// TIA Portal V15.1 export
// export: Created 2024-09-12T07:42:50.9677284Z, ExportSetting WithDefaults, DisplayName Totally Integrated Automation Portal, DisplayVersion V15.1 Update 5, DisplayName TIA Portal Openness, DisplayVersion V15.1 Update 5, DisplayName SINAMICS Startdrive Advanced, DisplayVersion V15.1, DisplayName G130, G150, S120, S150, SINAMICS MV, S210, DisplayVersion V15.1, DisplayName G110M, G120, G120C, G120D, G120P, DisplayVersion V15.1, DisplayName STEP 7 Professional, DisplayVersion V15.1 Update 5, DisplayName STEP 7 Safety, DisplayVersion V15.1, DisplayName WinCC Professional, DisplayVersion V15.1 Update 5, DisplayName SIMATIC Visualization Architect, DisplayVersion V15.1
FUNCTION_BLOCK "LSystemVarS7-1500"   // FB2204, FBD
TITLE = LSystemVarS7-1500
{ S7_Optimized_Access := 'TRUE' }
AUTHOR : VCC
FAMILY : Control
VERSION : 0.1
// =============================================================================
// This module is used to handle system variables such as Blink, Pulse, 
// ,Cycletime and CPU System Time used in timer modules.
// =============================================================================
// stored: AutoNumber false, IsIECCheckEnabled false, IsRetainMemResEnabled false, MemoryReserve 100, SetENOAutomatically False, UDAEnableTagReadback false
   VAR_INPUT
      I_OB1Cycletime { ExternalAccessible := 'False'; ExternalVisible := 'False'; ExternalWritable := 'False'} : Int;   // Cycle time of previous OB1 scan (milliseconds)
      I_PLCLADDR { ExternalAccessible := 'False'; ExternalVisible := 'False'; ExternalWritable := 'False'} : HW_IO;   // Hardware I/O
      I_DateTime { ExternalAccessible := 'False'; ExternalVisible := 'False'; ExternalWritable := 'False'} : Date_And_Time;   // Date and time
      I_AlarmResetPB { ExternalAccessible := 'False'; ExternalVisible := 'False'; ExternalWritable := 'False'} : Bool;   // Alarm reset pushbutton is activated / Alarm Reset Pushbutton is Activated
      I_EnableAlarm { ExternalAccessible := 'False'; ExternalVisible := 'False'; ExternalWritable := 'False'} : Bool := TRUE;   // Enable alarm from upper level / Enable Alarm from upper level
      C_HMIBtnResetSeqResetTM { ExternalAccessible := 'False'; ExternalVisible := 'False'; ExternalWritable := 'False'} : Bool;   // HMI buttons ResetSeq & ResetTM (0=Buttons are separate ; 1=Buttons are common)
      C_PlantId { ExternalAccessible := 'False'; ExternalVisible := 'False'; ExternalWritable := 'False'} : Int;   // Plant Identification (1=VCT, 2=VCBC, 3=VCG, 4=VCCH, 5=VCCD, 6=VCDQ, 7=AELQ, 8=PSCD)
      C_ShopId { ExternalAccessible := 'False'; ExternalVisible := 'False'; ExternalWritable := 'False'} : Int;   // Shop Identification (10=A-shop, 11=B-shop, 12=C-shop, 13=D-shop, 19=Stamping)
      C_LanguageChangeTimeToDefault { ExternalAccessible := 'False'; ExternalVisible := 'False'; ExternalWritable := 'False'} : Time := T#60m;   // Time to change back to default language. Connect T#0M to disable timer
   END_VAR
   VAR_OUTPUT
      O_AlarmABCondition { ExternalAccessible := 'False'; ExternalVisible := 'False'; ExternalWritable := 'False'} : Bool;   // Alarm AB condition / Alarm AB Condition
      O_AlarmA { ExternalAccessible := 'False'; ExternalVisible := 'False'; ExternalWritable := 'False'} : Bool;   // Summation Alarm A. / Alarm A
      O_AlarmB { ExternalAccessible := 'False'; ExternalVisible := 'False'; ExternalWritable := 'False'} : Bool;   // Summation Alarm B. / Alarm B
      O_AlarmC { ExternalAccessible := 'False'; ExternalVisible := 'False'; ExternalWritable := 'False'} : Bool;   // Summation Alarm C. / Alarm C.
      O_AlarmD { ExternalAccessible := 'False'; ExternalVisible := 'False'; ExternalWritable := 'False'} : Bool;   // Summation Alarm D. / Alarm D.
      O_AlarmWord { ExternalAccessible := 'False'; ExternalVisible := 'False'; ExternalWritable := 'False'} : DWord;   // Alarm Word
      O_SystemTime { ExternalAccessible := 'False'; ExternalVisible := 'False'; ExternalWritable := 'False'} : Array[0..2] of DWord;   // System Time
   END_VAR
   VAR_IN_OUT
      IO_Alarm : "Alarm";   // Alarm
      IO_SetDateTime { ExternalAccessible := 'False'; ExternalVisible := 'False'; ExternalWritable := 'False'} : Bool;   // Set date and time
      H_HMI : "H_HMI";   // HMI
      "H_SystemVarS7-1500" : "H_SystemVarS7-1500";   // Animation
      C_SwedishLanguage { ExternalAccessible := 'False'; ExternalVisible := 'False'; ExternalWritable := 'False'} : Bool;   // Swedisch Language
      C_DutchLanguage { ExternalAccessible := 'False'; ExternalVisible := 'False'; ExternalWritable := 'False'} : Bool;   // Dutch Language
      C_EnglishLanguage { ExternalAccessible := 'False'; ExternalVisible := 'False'; ExternalWritable := 'False'} : Bool;   // English Language
      C_ChineseLanguage { ExternalAccessible := 'False'; ExternalVisible := 'False'; ExternalWritable := 'False'} : Bool;   // Chinese Language
      C_ScreenSaverEnable { ExternalAccessible := 'False'; ExternalVisible := 'False'; ExternalWritable := 'False'} : Bool;   // Screen Saver HMI Panels
   END_VAR
   VAR
      AB_FALSE { ExternalAccessible := 'False'; ExternalVisible := 'False'; ExternalWritable := 'False'} : Bool;   // Systemvariabel Logiskt Resultat "TRUE" = "FALSE" / System Variable Logic Result TRUE Should Be FALSE
      AB_TRUE { ExternalAccessible := 'False'; ExternalVisible := 'False'; ExternalWritable := 'False'} : Bool;   // Systemvariabel Logiskt Resultat "FALSE" = "TRUE" / System Variable Logic Result FALSE Should Be TRUE
      AD_OB40 { ExternalAccessible := 'False'; ExternalVisible := 'False'; ExternalWritable := 'False'} : Bool;   // 0000: Hardware Interrupt 0 / Hardware Interrupt / Hårdvaru Interrupt
      AD_OB80 { ExternalAccessible := 'False'; ExternalVisible := 'False'; ExternalWritable := 'False'} : Bool;   // 0000: Cycle Time Fault / Cycle Time Error / Cykeltidsfel
      AD_OB81 { ExternalAccessible := 'False'; ExternalVisible := 'False'; ExternalWritable := 'False'} : Bool;   // 0000: Power Supply Fault / Error On Power Supply / Fel På Spänningsaggregat
      AD_OB82 { ExternalAccessible := 'False'; ExternalVisible := 'False'; ExternalWritable := 'False'} : Bool;   // 0000: I/O Point Fault 1 / I/O Error / I/O Fel
      AD_OB83 { ExternalAccessible := 'False'; ExternalVisible := 'False'; ExternalWritable := 'False'} : Bool;   // 0000: I/O Point Fault 2 / I/O Error / I/O Fel
      AD_OB84 { ExternalAccessible := 'False'; ExternalVisible := 'False'; ExternalWritable := 'False'} : Bool;   // 0000: CPU Fault / CPU Error / CPU Fel
      AD_OB85 { ExternalAccessible := 'False'; ExternalVisible := 'False'; ExternalWritable := 'False'} : Bool;   // 0000: OB Not Loaded Fault / I/O Access Error / I/O Access Fel
      AD_OB86 { ExternalAccessible := 'False'; ExternalVisible := 'False'; ExternalWritable := 'False'} : Bool;   // 0000: Loss of Rack Fault / CPU Rack Error / CPU Rack Fel
      AD_OB87 { ExternalAccessible := 'False'; ExternalVisible := 'False'; ExternalWritable := 'False'} : Bool;   // 0000: Communication Fault / Communication Error / Kommunikationsfel
      AD_OB100 { ExternalAccessible := 'False'; ExternalVisible := 'False'; ExternalWritable := 'False'} : Bool;   // 0000: Complete Restart / CPU Warm Restart / CPU Varm Omstart
      AD_OB101 { ExternalAccessible := 'False'; ExternalVisible := 'False'; ExternalWritable := 'False'} : Bool;   // Hot Restart / Omstart
      AD_OB102 { ExternalAccessible := 'False'; ExternalVisible := 'False'; ExternalWritable := 'False'} : Bool;   // 0000: Cold Restart / Cold Restart / Omstart
      AB_OB121 { ExternalAccessible := 'False'; ExternalVisible := 'False'; ExternalWritable := 'False'} : Bool;   // 0000: Programming Error / Programming Error / Programmeringsfel
      AD_OB122 { ExternalAccessible := 'False'; ExternalVisible := 'False'; ExternalWritable := 'False'} : Bool;   // 0000: Module Access Error / I/O Module Access Error / I/O Modul Access Fel
      AD_Forced { ExternalAccessible := 'False'; ExternalVisible := 'False'; ExternalWritable := 'False'} : Bool;   // 0000: Forced I/O in CPU / I/O Are Forced In CPU / I/O Är Forcerade I CPU
      AD_Error { ExternalAccessible := 'False'; ExternalVisible := 'False'; ExternalWritable := 'False'} : Bool;   // Error In Software Or Hardware Check Diagnostics / Fel I Mjukvara Eller Hårdvara Kontrollera Diagnostik
      AD_Warning { ExternalAccessible := 'False'; ExternalVisible := 'False'; ExternalWritable := 'False'} : Bool;   // Warning In Software Or Hardware Check Diagnostics / Varning I Mjukvara Eller Hårdvara Kontrollera Diagnostik
      AE_CalibrationMovUnit { ExternalAccessible := 'False'; ExternalVisible := 'False'; ExternalWritable := 'False'} : Bool;   // Kalibrering MovUnit's Utförd / Info -> Redo Overtime calibration MovUnit / Calibration MovUnit's Executed
      AE_CalibrationTransfers { ExternalAccessible := 'False'; ExternalVisible := 'False'; ExternalWritable := 'False'} : Bool;   // Kalibrering MovUnit's Utförd / Info -> Redo Overtime calibration Transfers / Calibration MovUnit's Executed
      AE_Simulation { ExternalAccessible := 'False'; ExternalVisible := 'False'; ExternalWritable := 'False'} : Bool;   // Kalibrering MovUnit's Utförd / Info -> Simulation is active / Calibration MovUnit's Executed
      PulseBlink0_1s { ExternalAccessible := 'False'; ExternalVisible := 'False'; ExternalWritable := 'False'} : Bool;   // Help memory for pulse 0.1s
      PulseBlink0_2s { ExternalAccessible := 'False'; ExternalVisible := 'False'; ExternalWritable := 'False'} : Bool;   // Help memory for pulse 0.2s
      PulseBlink0_4s { ExternalAccessible := 'False'; ExternalVisible := 'False'; ExternalWritable := 'False'} : Bool;   // Help memory for pulse 0.4s
      PulseBlink0_5s { ExternalAccessible := 'False'; ExternalVisible := 'False'; ExternalWritable := 'False'} : Bool;   // Help memory for pulse 0.5s
      PulseBlink0_8s { ExternalAccessible := 'False'; ExternalVisible := 'False'; ExternalWritable := 'False'} : Bool;   // Help memory for pulse 0.8s
      PulseBlink1_0s { ExternalAccessible := 'False'; ExternalVisible := 'False'; ExternalWritable := 'False'} : Bool;   // Help memory for pulse 1.0s
      PulseBlink1_6s { ExternalAccessible := 'False'; ExternalVisible := 'False'; ExternalWritable := 'False'} : Bool;   // Help memory for pulse 1.6s
      PulseBlink2_0s { ExternalAccessible := 'False'; ExternalVisible := 'False'; ExternalWritable := 'False'} : Bool;   // Help memory for pulse 2.0s
      AlarmA { ExternalAccessible := 'False'; ExternalVisible := 'False'; ExternalWritable := 'False'} : Bool;   // Summation Alarm A / Alarm A
      AlarmB { ExternalAccessible := 'False'; ExternalVisible := 'False'; ExternalWritable := 'False'} : Bool;   // Summation Alarm B / Alarm B
      AlarmC { ExternalAccessible := 'False'; ExternalVisible := 'False'; ExternalWritable := 'False'} : Bool;   // Summation Alarm C / Alarm C
      AlarmD { ExternalAccessible := 'False'; ExternalVisible := 'False'; ExternalWritable := 'False'} : Bool;   // Summation Alarm D / Alarm D
      AlarmOB40 { ExternalAccessible := 'False'; ExternalVisible := 'False'; ExternalWritable := 'False'} : Bool;   // Alarm OB40
      AlarmOB80 { ExternalAccessible := 'False'; ExternalVisible := 'False'; ExternalWritable := 'False'} : Bool;   // Alarm OB80
      AlarmOB81 { ExternalAccessible := 'False'; ExternalVisible := 'False'; ExternalWritable := 'False'} : Bool;   // Alarm OB81
      AlarmOB82 { ExternalAccessible := 'False'; ExternalVisible := 'False'; ExternalWritable := 'False'} : Bool;   // Alarm OB82
      AlarmOB83 { ExternalAccessible := 'False'; ExternalVisible := 'False'; ExternalWritable := 'False'} : Bool;   // Alarm OB83
      AlarmOB84 { ExternalAccessible := 'False'; ExternalVisible := 'False'; ExternalWritable := 'False'} : Bool;   // Alarm OB84
      AlarmOB85 { ExternalAccessible := 'False'; ExternalVisible := 'False'; ExternalWritable := 'False'} : Bool;   // Alarm OB85
      AlarmOB86 { ExternalAccessible := 'False'; ExternalVisible := 'False'; ExternalWritable := 'False'} : Bool;   // Alarm OB86
      AlarmOB87 { ExternalAccessible := 'False'; ExternalVisible := 'False'; ExternalWritable := 'False'} : Bool;   // Alarm OB87
      AlarmOB100 { ExternalAccessible := 'False'; ExternalVisible := 'False'; ExternalWritable := 'False'} : Bool;   // Alarm OB100
      AlarmOB101 { ExternalAccessible := 'False'; ExternalVisible := 'False'; ExternalWritable := 'False'} : Bool;   // Alarm OB101
      AlarmOB102 { ExternalAccessible := 'False'; ExternalVisible := 'False'; ExternalWritable := 'False'} : Bool;   // Alarm OB102
      AlarmOB121 { ExternalAccessible := 'False'; ExternalVisible := 'False'; ExternalWritable := 'False'} : Bool;   // Alarm OB121
      AlarmOB122 { ExternalAccessible := 'False'; ExternalVisible := 'False'; ExternalWritable := 'False'} : Bool;   // Alarm OB122
      Edge { ExternalAccessible := 'False'; ExternalVisible := 'False'; ExternalWritable := 'False'} : Array[0..15] of Bool;   // Edge
      MemOB40Execution { ExternalAccessible := 'False'; ExternalVisible := 'False'; ExternalWritable := 'False'} : Int;   // Memorisation previous value number of executuons of OB40
      MemOB80Execution { ExternalAccessible := 'False'; ExternalVisible := 'False'; ExternalWritable := 'False'} : Int;   // Memorisation previous value number of executuons of OB80
      MemOB81Execution { ExternalAccessible := 'False'; ExternalVisible := 'False'; ExternalWritable := 'False'} : Int;   // Memorisation previous value number of executuons of OB81
      MemOB82Execution { ExternalAccessible := 'False'; ExternalVisible := 'False'; ExternalWritable := 'False'} : Int;   // Memorisation previous value number of executuons of OB82
      MemOB83Execution { ExternalAccessible := 'False'; ExternalVisible := 'False'; ExternalWritable := 'False'} : Int;   // Memorisation previous value number of executuons of OB83
      MemOB84Execution { ExternalAccessible := 'False'; ExternalVisible := 'False'; ExternalWritable := 'False'} : Int;   // Memorisation previous value number of executuons of OB84
      MemOB85Execution { ExternalAccessible := 'False'; ExternalVisible := 'False'; ExternalWritable := 'False'} : Int;   // Memorisation previous value number of executuons of OB85
      MemOB86Execution { ExternalAccessible := 'False'; ExternalVisible := 'False'; ExternalWritable := 'False'} : Int;   // Memorisation previous value number of executuons of OB86
      MemOB87Execution { ExternalAccessible := 'False'; ExternalVisible := 'False'; ExternalWritable := 'False'} : Int;   // Memorisation previous value number of executuons of OB87
      MemOB100Execution { ExternalAccessible := 'False'; ExternalVisible := 'False'; ExternalWritable := 'False'} : Int;   // Memorisation previous value number of executuons of OB100
      MemOB101Execution { ExternalAccessible := 'False'; ExternalVisible := 'False'; ExternalWritable := 'False'} : Int;   // Memorisation previous value number of executuons of OB101
      MemOB102Execution { ExternalAccessible := 'False'; ExternalVisible := 'False'; ExternalWritable := 'False'} : Int;   // Memorisation previous value number of executuons of OB102
      MemOB121Execution { ExternalAccessible := 'False'; ExternalVisible := 'False'; ExternalWritable := 'False'} : Int;   // Memorisation previous value number of executuons of OB121
      MemOB122Execution { ExternalAccessible := 'False'; ExternalVisible := 'False'; ExternalWritable := 'False'} : Int;   // Memorisation previous value number of executuons of OB122
      HMICmd_CalibrateMovUnits { ExternalAccessible := 'False'; ExternalVisible := 'False'; ExternalWritable := 'False'} : Bool;   // HMI Command - Calibrate Move Units
      HMICmd_CalibrateTransfers { ExternalAccessible := 'False'; ExternalVisible := 'False'; ExternalWritable := 'False'} : Bool;   // HMI Command - Calibrate Transfers
      HMICmd_Simulation { ExternalAccessible := 'False'; ExternalVisible := 'False'; ExternalWritable := 'False'} : Bool;   // HMI Command - Simulation
      HMICmd_DisableIOAlarm { ExternalAccessible := 'False'; ExternalVisible := 'False'; ExternalWritable := 'False'} : Bool;   // HMI Command - Disable IO Alarm
      ActualScanTimeOB1 { ExternalAccessible := 'False'; ExternalVisible := 'False'; ExternalWritable := 'False'} : LTime;   // Animation / FB
      LongestScanTimeOB1 { ExternalAccessible := 'False'; ExternalVisible := 'False'; ExternalWritable := 'False'} : LTime;   // Animation / FB
      EnableAlarm { ExternalAccessible := 'False'; ExternalVisible := 'False'; ExternalWritable := 'False'} : Bool := TRUE;   // Enable alarm from upper level / Enable Alarm from upper level
      LanguageChangeToDefault { ExternalAccessible := 'False'; ExternalVisible := 'False'; ExternalWritable := 'False'} : Bool;   // Change language back to default
      LanguageDefaultTime { ExternalAccessible := 'False'; ExternalVisible := 'False'; ExternalWritable := 'False'} : DInt;   // Language to default time running value
      DBnr { ExternalAccessible := 'False'; ExternalVisible := 'False'; ExternalWritable := 'False'} : Int;   // HMI DB number
      TimerOffOB40 { ExternalAccessible := 'False'; ExternalVisible := 'False'; ExternalWritable := 'False'} : TOF_TIME;   // FB / Timer
      TimerOffOB80 { ExternalAccessible := 'False'; ExternalVisible := 'False'; ExternalWritable := 'False'} : TOF_TIME;   // FB / Timer
      TimerOffOB81 { ExternalAccessible := 'False'; ExternalVisible := 'False'; ExternalWritable := 'False'} : TOF_TIME;   // FB / Timer
      TimerOffB83 { ExternalAccessible := 'False'; ExternalVisible := 'False'; ExternalWritable := 'False'} : TOF_TIME;   // FB / Timer
      TimerOffOB84 { ExternalAccessible := 'False'; ExternalVisible := 'False'; ExternalWritable := 'False'} : TOF_TIME;   // FB / Timer
      TimerOffOB85 { ExternalAccessible := 'False'; ExternalVisible := 'False'; ExternalWritable := 'False'} : TOF_TIME;   // FB / Timer
      TimerOffOB86 { ExternalAccessible := 'False'; ExternalVisible := 'False'; ExternalWritable := 'False'} : TOF_TIME;   // FB / Timer
      TimerOffOB87 { ExternalAccessible := 'False'; ExternalVisible := 'False'; ExternalWritable := 'False'} : TOF_TIME;   // FB / Timer
      TimerOffOB100 { ExternalAccessible := 'False'; ExternalVisible := 'False'; ExternalWritable := 'False'} : TOF_TIME;   // FB / Timer
      TimerOffOB101 { ExternalAccessible := 'False'; ExternalVisible := 'False'; ExternalWritable := 'False'} : TOF_TIME;   // FB / Timer
      TimerOffOB102 { ExternalAccessible := 'False'; ExternalVisible := 'False'; ExternalWritable := 'False'} : TOF_TIME;   // FB / Timer
      TimerOffOB121 { ExternalAccessible := 'False'; ExternalVisible := 'False'; ExternalWritable := 'False'} : TOF_TIME;   // FB / Timer
      TimerOffOB122 { ExternalAccessible := 'False'; ExternalVisible := 'False'; ExternalWritable := 'False'} : TOF_TIME;   // FB / Timer
      TimerCalibrationMovUnit { ExternalAccessible := 'False'; ExternalVisible := 'False'; ExternalWritable := 'False'} : TOF_TIME;   // Timer
      TimerCalibrationTransfers { ExternalAccessible := 'False'; ExternalVisible := 'False'; ExternalWritable := 'False'} : TOF_TIME;   // Timer
      TimerGlobalSelAutoMode { ExternalAccessible := 'False'; ExternalVisible := 'False'; ExternalWritable := 'False'} : TON_TIME;   // Timer
      TimerGlobalSelManualMode { ExternalAccessible := 'False'; ExternalVisible := 'False'; ExternalWritable := 'False'} : TON_TIME;   // Timer
      _GetIMData { ExternalAccessible := 'False'; ExternalVisible := 'False'; ExternalWritable := 'False'} : Get_IM_Data;   // FB
      _DlyErr { ExternalAccessible := 'False'; ExternalVisible := 'False'; ExternalWritable := 'False'} : TON_TIME;   // Timer
      _DlyWarning { ExternalAccessible := 'False'; ExternalVisible := 'False'; ExternalWritable := 'False'} : TON_TIME;   // Timer
      _ScreenSaverHMI { ExternalAccessible := 'False'; ExternalVisible := 'False'; ExternalWritable := 'False'} : "LTimer";   // Timer
      _LanguageDefault { ExternalAccessible := 'False'; ExternalVisible := 'False'; ExternalWritable := 'False'} : TON_TIME;   // Timer
      _LToggleDisableIOAlarm { ExternalAccessible := 'False'; ExternalVisible := 'False'; ExternalWritable := 'False'} : "LToggle";   // FB
   END_VAR
   VAR_TEMP
      TmpSystemTime : DTL;   // Temporary DTL Day / Temp
      TmpSystemHourMin : UInt;   // Temp
      TmpRetValTime : Int;   // Temp RetVal of TD_SYS_T / Temp
      TmpWeekday : Int;   // Temporary weekday / Temp
      TmpResult : Int;   // Temporary result / Temp
      SetClkRet : Int;   // Return value / Temp
      ReadSysstData : Struct   // data read / Temp
         "STOP/RUN" : Int;   // Stop, Run
         ERROR : Int;   // Error
         MAINT : Int;   // Maintanance
      END_STRUCT;
      LED1C1On : Bool;   // LED 1 color 1: Green on
      LED1C1Blink : Bool;   // LED 1 color 1: Green blinking
      LED1C2On : Bool;   // LED 1 color 2: Yellow on
      LED1C2Blink : Bool;   // LED 1 color 2: Yellow blinking
      LED2C1On : Bool;   // LED 2 color 1: Red on
      LED2C1Blink : Bool;   // LED 2 color 1: Red blinking
      LED3C1On : Bool;   // LED 3 color 1: Yellow on
      LED3C1Blink : Bool;   // LED 3 color 1: Yellow blinking
      IMData : IM0_Data;   // Temp
      tNotUsedDInt : DInt;   // Temp
   END_VAR
   VAR_TEMP   // added for the SCL form of the ladder/FBD networks
      _w1 : Bool;
      _w2 : Bool;
      _w3 : Bool;
      _w4 : Bool;
      _w5 : Bool;
   END_VAR
BEGIN

REGION Network 1: **** 1 - Inputs **** Extract HMI Commands
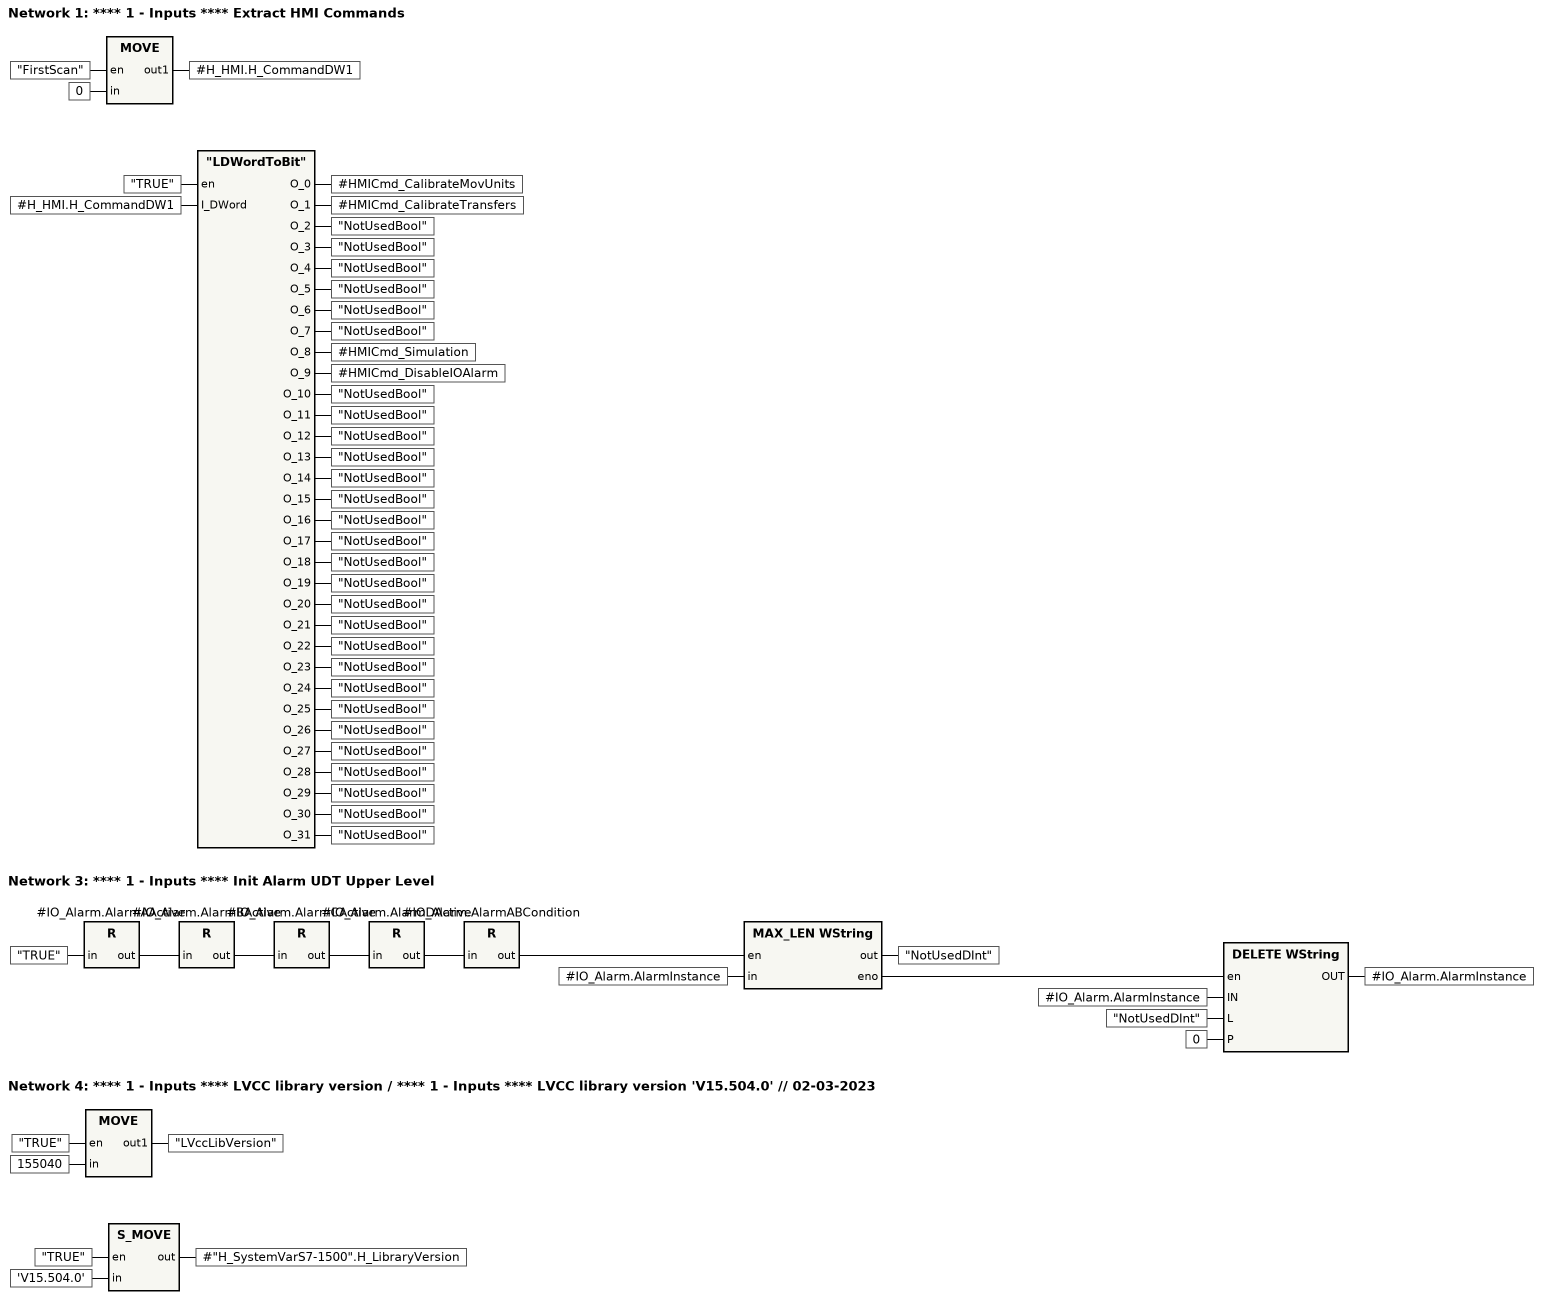
   IF "FirstScan" THEN #H_HMI.H_CommandDW1 := 0; END_IF;
   IF "TRUE" THEN
       "LDWordToBit"(I_DWord := #H_HMI.H_CommandDW1,
                     O_0 => #HMICmd_CalibrateMovUnits,
                     O_1 => #HMICmd_CalibrateTransfers,
                     O_2 => "NotUsedBool",
                     O_3 => "NotUsedBool",
                     O_4 => "NotUsedBool",
                     O_5 => "NotUsedBool",
                     O_6 => "NotUsedBool",
                     O_7 => "NotUsedBool",
                     O_8 => #HMICmd_Simulation,
                     O_9 => #HMICmd_DisableIOAlarm,
                     O_10 => "NotUsedBool",
                     O_11 => "NotUsedBool",
                     O_12 => "NotUsedBool",
                     O_13 => "NotUsedBool",
                     O_14 => "NotUsedBool",
                     O_15 => "NotUsedBool",
                     O_16 => "NotUsedBool",
                     O_17 => "NotUsedBool",
                     O_18 => "NotUsedBool",
                     O_19 => "NotUsedBool",
                     O_20 => "NotUsedBool",
                     O_21 => "NotUsedBool",
                     O_22 => "NotUsedBool",
                     O_23 => "NotUsedBool",
                     O_24 => "NotUsedBool",
                     O_25 => "NotUsedBool",
                     O_26 => "NotUsedBool",
                     O_27 => "NotUsedBool",
                     O_28 => "NotUsedBool",
                     O_29 => "NotUsedBool",
                     O_30 => "NotUsedBool",
                     O_31 => "NotUsedBool");
   END_IF;
END_REGION

NETWORK
TITLE = **** 1 - Inputs **** DB number
// DB number
      L     DINO;
      T     #DBnr;

REGION Network 3: **** 1 - Inputs **** Init Alarm UDT Upper Level
   // Alarm / Alarm D / Init Alarm UDT Upper Level
   // ENO of a box is taken as its EN; it also drops when the box reports an error
   IF "TRUE" THEN
       #IO_Alarm.AlarmAActive := FALSE;
       #IO_Alarm.AlarmBActive := FALSE;
       #IO_Alarm.AlarmCActive := FALSE;
       #IO_Alarm.AlarmDActive := FALSE;
       #IO_Alarm.AlarmABCondition := FALSE;
   END_IF;
   #_w1 := "TRUE";
   IF #_w1 THEN
       MAX_LEN(in := #IO_Alarm.AlarmInstance, out => "NotUsedDInt");
       DELETE(IN := #IO_Alarm.AlarmInstance, L := "NotUsedDInt", P := 0, OUT => #IO_Alarm.AlarmInstance);
   END_IF;
END_REGION

REGION Network 4: **** 1 - Inputs **** LVCC library version / **** 1 - Inputs **** LVCC library version 'V15.504.0' // 02-03-2023
   // LVCC library version
   IF "TRUE" THEN
       "LVccLibVersion" := 155040;
       #"H_SystemVarS7-1500".H_LibraryVersion := 'V15.504.0';
   END_IF;
END_REGION

NETWORK
TITLE = **** 1 - Inputs **** Load Constants
// Load Constants
      L     1;
      T     "1Ms";
      L     50;
      T     "50Ms";
      L     100;
      T     "100Ms";
      L     500;
      T     "500Ms";
      L     1000;
      T     "1000Ms";
      L     5000;
      T     "5000Ms";
      L     10000;
      T     "10000Ms";
      L     0;
      T     "Zero";
      NOP   0;
//Init Calibrate Mov Units 1 Scan
      A     #HMICmd_CalibrateMovUnits;
      FP    #Edge[0];
      =     "CalibrateMovUnits";
//Init Calibrate Transfers 1 Scan
      A     #HMICmd_CalibrateTransfers;
      FP    #Edge[3];
      =     "CalibrateTransfer";


REGION Network 6: **** 1 - Inputs **** Disable IO_Alarm
   // Disable IO_Alarm
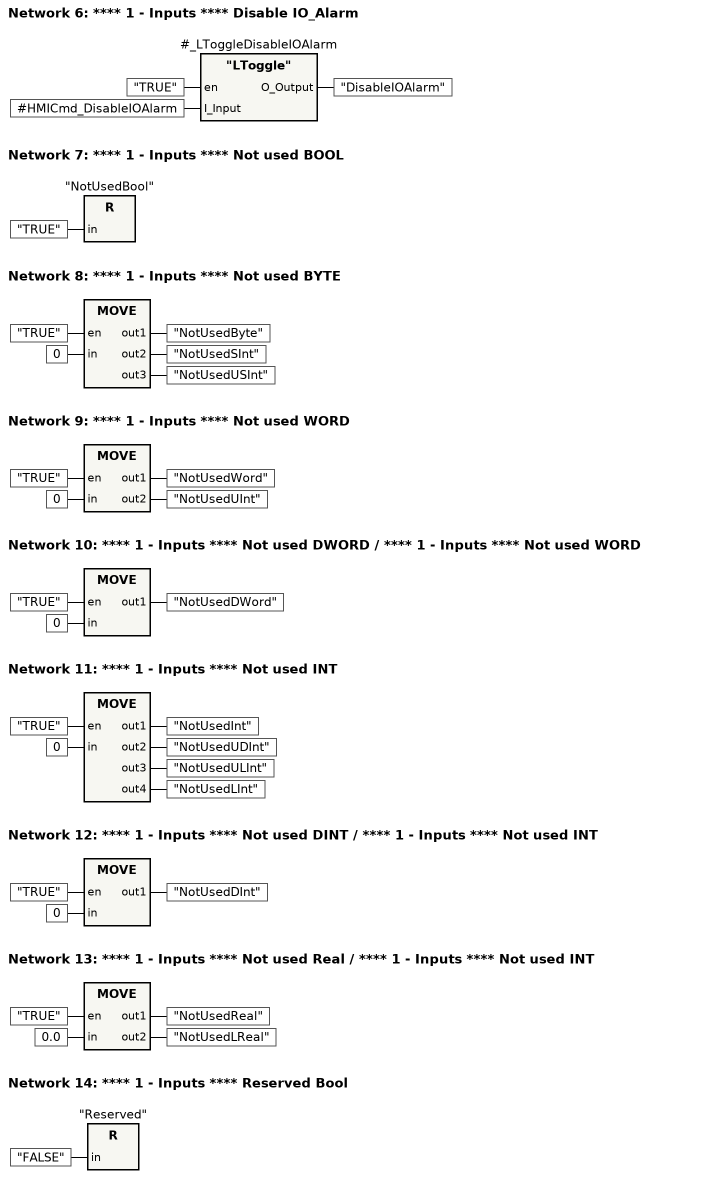
   IF "TRUE" THEN
       #_LToggleDisableIOAlarm(I_Input := #HMICmd_DisableIOAlarm, O_Output => "DisableIOAlarm");   // "LToggle"
   END_IF;
END_REGION

REGION Network 7: **** 1 - Inputs **** Not used BOOL
   // Not used BOOL
   IF "TRUE" THEN "NotUsedBool" := FALSE; END_IF;
END_REGION

REGION Network 8: **** 1 - Inputs **** Not used BYTE
   // Not used BYTE
   IF "TRUE" THEN
       "NotUsedByte" := 0;
       "NotUsedSInt" := 0;
       "NotUsedUSInt" := 0;
   END_IF;
END_REGION

REGION Network 9: **** 1 - Inputs **** Not used WORD
   // Not used WORD
   IF "TRUE" THEN
       "NotUsedWord" := 0;
       "NotUsedUInt" := 0;
   END_IF;
END_REGION

REGION Network 10: **** 1 - Inputs **** Not used DWORD / **** 1 - Inputs **** Not used WORD
   // Not used DWORD / Not used WORD
   IF "TRUE" THEN "NotUsedDWord" := 0; END_IF;
END_REGION

REGION Network 11: **** 1 - Inputs **** Not used INT
   // Not used INT
   IF "TRUE" THEN
       "NotUsedInt" := 0;
       "NotUsedUDInt" := 0;
       "NotUsedULInt" := 0;
       "NotUsedLInt" := 0;
   END_IF;
END_REGION

REGION Network 12: **** 1 - Inputs **** Not used DINT / **** 1 - Inputs **** Not used INT
   // Not used DINT / Not used INT
   IF "TRUE" THEN "NotUsedDInt" := 0; END_IF;
END_REGION

REGION Network 13: **** 1 - Inputs **** Not used Real / **** 1 - Inputs **** Not used INT
   // Not used DINT / Not used INT
   IF "TRUE" THEN
       "NotUsedReal" := 0.0;
       "NotUsedLReal" := 0.0;
   END_IF;
END_REGION

REGION Network 14: **** 1 - Inputs **** Reserved Bool
   // Reserverd for HMI functionality
   IF "FALSE" THEN "Reserved" := FALSE; END_IF;
END_REGION

REGION Network 15: **** 1 - Inputs **** Load Language In HMI
   // Load Language In HMI / Not used INT
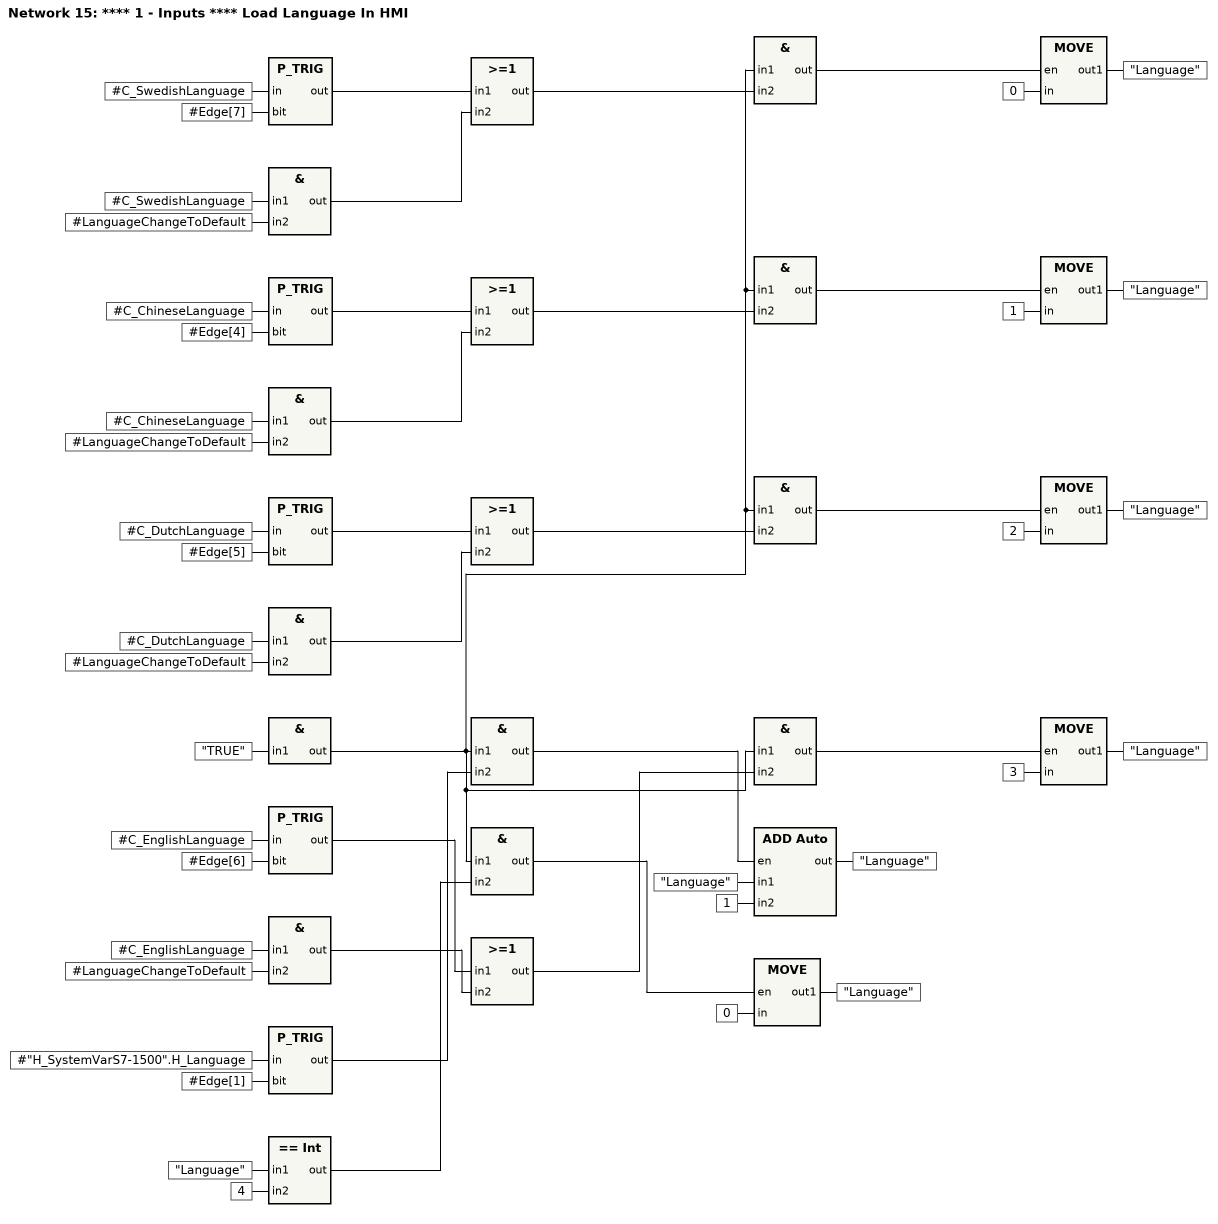
   #_w1 := #C_SwedishLanguage AND NOT #Edge[7];   // rising edge
   #Edge[7] := #C_SwedishLanguage;
   IF "TRUE" AND (#_w1 OR (#C_SwedishLanguage AND #LanguageChangeToDefault)) THEN "Language" := 0; END_IF;
   #_w2 := #C_ChineseLanguage AND NOT #Edge[4];   // rising edge
   #Edge[4] := #C_ChineseLanguage;
   IF "TRUE" AND (#_w2 OR (#C_ChineseLanguage AND #LanguageChangeToDefault)) THEN "Language" := 1; END_IF;
   #_w3 := #C_DutchLanguage AND NOT #Edge[5];   // rising edge
   #Edge[5] := #C_DutchLanguage;
   IF "TRUE" AND (#_w3 OR (#C_DutchLanguage AND #LanguageChangeToDefault)) THEN "Language" := 2; END_IF;
   #_w4 := #C_EnglishLanguage AND NOT #Edge[6];   // rising edge
   #Edge[6] := #C_EnglishLanguage;
   IF "TRUE" AND (#_w4 OR (#C_EnglishLanguage AND #LanguageChangeToDefault)) THEN "Language" := 3; END_IF;
   #_w5 := #"H_SystemVarS7-1500".H_Language AND NOT #Edge[1];   // rising edge
   #Edge[1] := #"H_SystemVarS7-1500".H_Language;
   IF "TRUE" AND #_w5 THEN "Language" := "Language" + 1; END_IF;
   IF "TRUE" AND ("Language" = 4) THEN "Language" := 0; END_IF;
END_REGION

REGION Network 16: **** 1 - Inputs **** Simulation ON/OFF
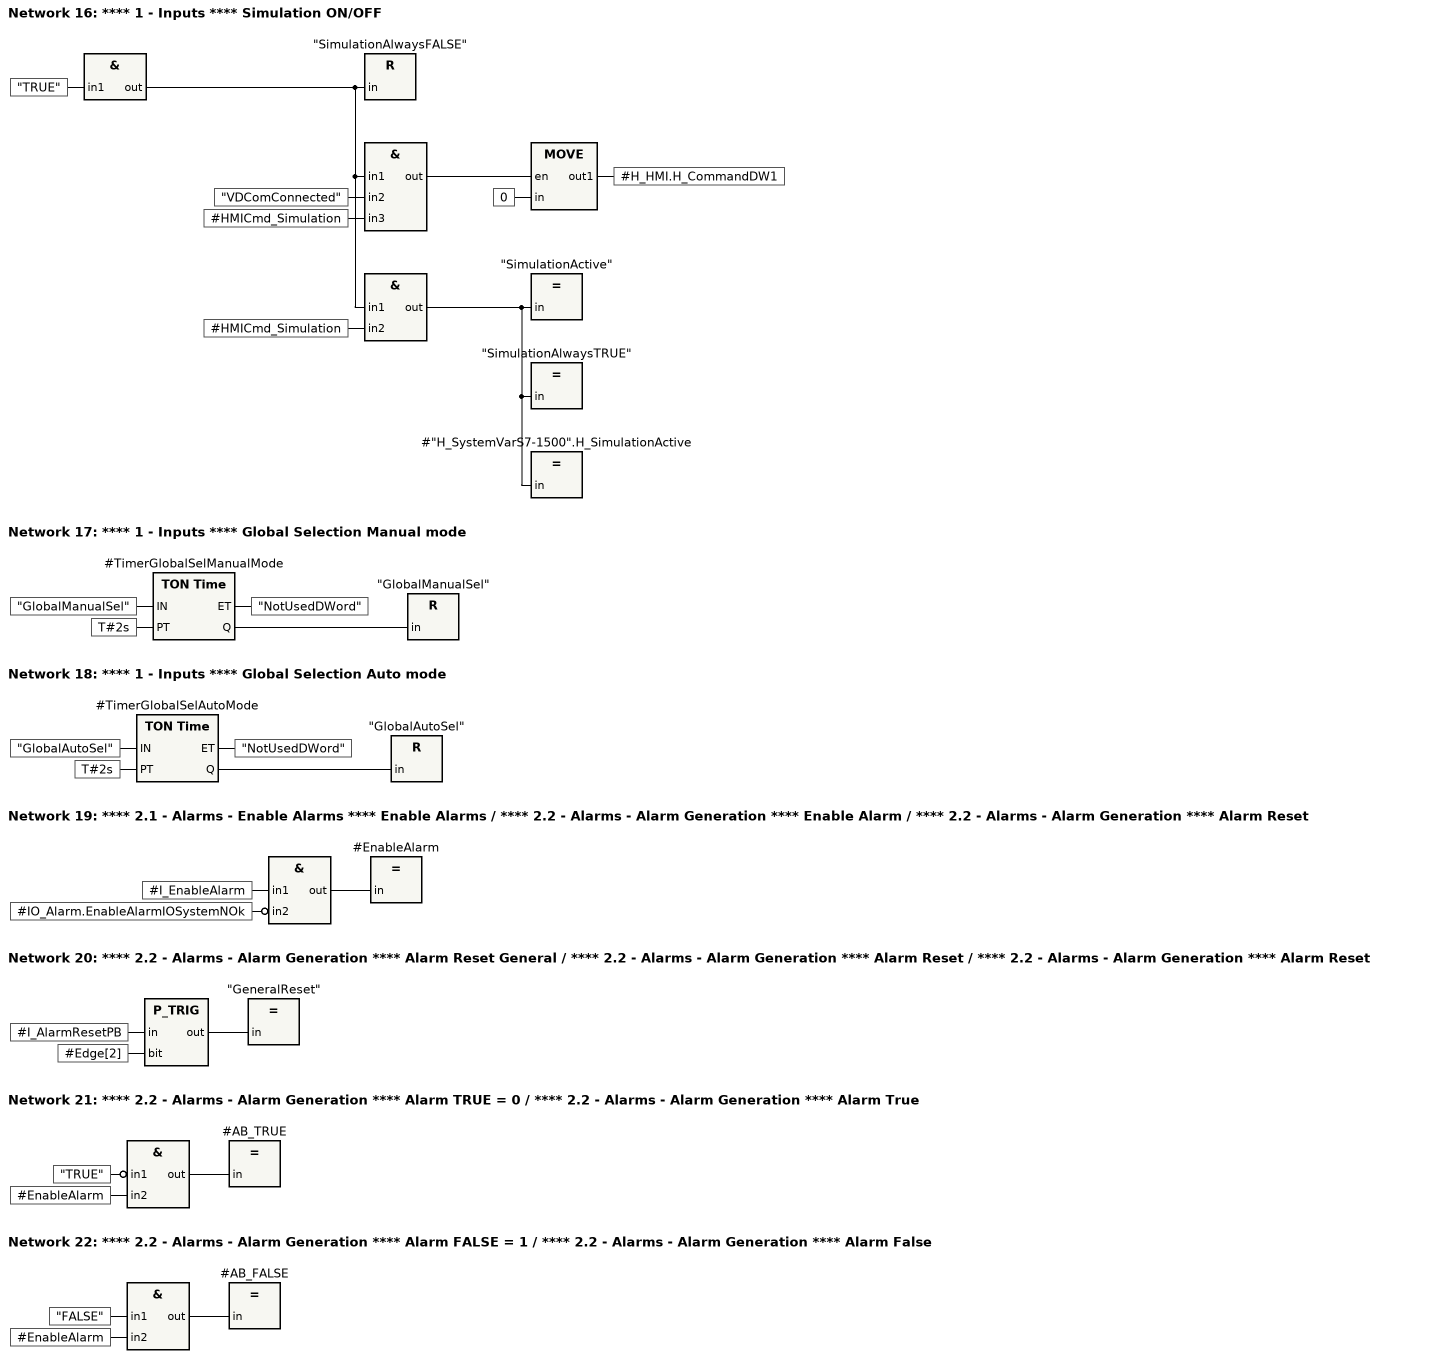
   IF "TRUE" THEN "SimulationAlwaysFALSE" := FALSE; END_IF;
   IF "TRUE" AND "VDComConnected" AND #HMICmd_Simulation THEN #H_HMI.H_CommandDW1 := 0; END_IF;
   "SimulationActive" := "TRUE" AND #HMICmd_Simulation;
   "SimulationAlwaysTRUE" := "SimulationActive";
   #"H_SystemVarS7-1500".H_SimulationActive := "SimulationActive";
END_REGION

REGION Network 17: **** 1 - Inputs **** Global Selection Manual mode
   #TimerGlobalSelManualMode(IN := "GlobalManualSel", PT := T#2s, ET => "NotUsedDWord");   // TON
   IF #TimerGlobalSelManualMode.Q THEN "GlobalManualSel" := FALSE; END_IF;
END_REGION

REGION Network 18: **** 1 - Inputs **** Global Selection Auto mode
   #TimerGlobalSelAutoMode(IN := "GlobalAutoSel", PT := T#2s, ET => "NotUsedDWord");   // TON
   IF #TimerGlobalSelAutoMode.Q THEN "GlobalAutoSel" := FALSE; END_IF;
END_REGION

REGION Network 19: **** 2.1 - Alarms - Enable Alarms **** Enable Alarms / **** 2.2 - Alarms - Alarm Generation **** Enable Alarm / **** 2.2 - Alarms - Alarm Generation **** Alarm Reset
   // Enable Alarms
   // Alarm Reset
   //  - via inputs
   //  - AutoReset Alarm C or Alarm D if no Alarm A or B present
   #EnableAlarm := #I_EnableAlarm AND NOT #IO_Alarm.EnableAlarmIOSystemNOk;
END_REGION

REGION Network 20: **** 2.2 - Alarms - Alarm Generation **** Alarm Reset General / **** 2.2 - Alarms - Alarm Generation **** Alarm Reset / **** 2.2 - Alarms - Alarm Generation **** Alarm Reset
   // Alarm Reset General
   // Alarm Reset
   //  - via inputs
   //  - AutoReset Alarm C or Alarm D if no Alarm A or B present
   // Alarm Reset
   #_w1 := #I_AlarmResetPB AND NOT #Edge[2];   // rising edge
   #Edge[2] := #I_AlarmResetPB;
   "GeneralReset" := #_w1;
END_REGION

REGION Network 21: **** 2.2 - Alarms - Alarm Generation **** Alarm TRUE = 0 / **** 2.2 - Alarms - Alarm Generation **** Alarm True
   // Alarm / Alarm Reset
   #AB_TRUE := NOT "TRUE" AND #EnableAlarm;
END_REGION

REGION Network 22: **** 2.2 - Alarms - Alarm Generation **** Alarm FALSE = 1 / **** 2.2 - Alarms - Alarm Generation **** Alarm False
   // Alarm
   // Alarm Reset
   //  - via inputs
   //  - AutoReset Alarm C or Alarm D if no Alarm A or B present
   #AB_FALSE := "FALSE" AND #EnableAlarm;
END_REGION

REGION Network 23: **** 2.2 - Alarms - Alarm Generation **** Alarm exception OB40
   // Alarm exception OB40
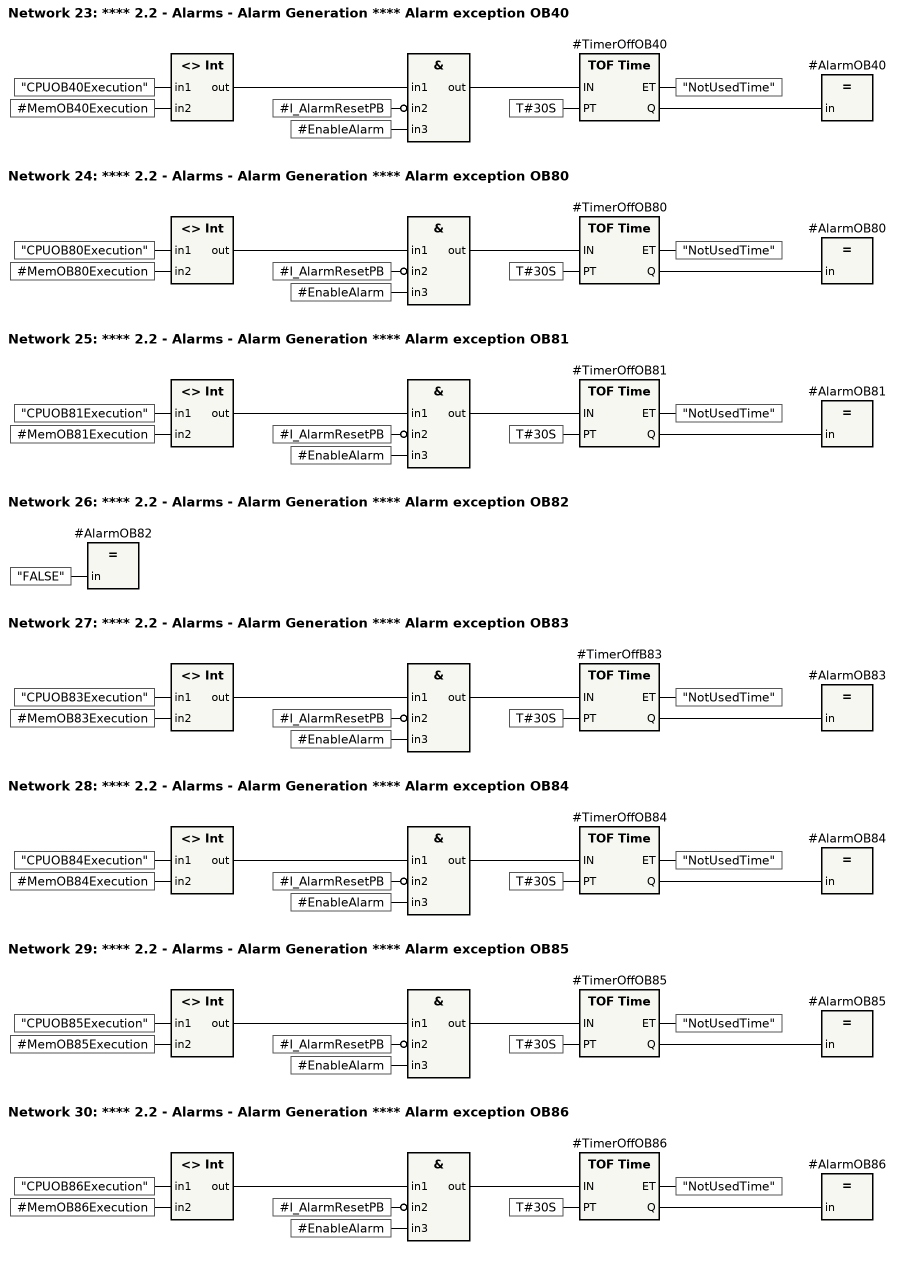
   #TimerOffOB40(IN := ("CPUOB40Execution" <> #MemOB40Execution) AND NOT #I_AlarmResetPB AND #EnableAlarm,   // TOF
                 PT := T#30S,
                 ET => "NotUsedTime");
   #AlarmOB40 := #TimerOffOB40.Q;
END_REGION

REGION Network 24: **** 2.2 - Alarms - Alarm Generation **** Alarm exception OB80
   // Alarm exception OB80
   #TimerOffOB80(IN := ("CPUOB80Execution" <> #MemOB80Execution) AND NOT #I_AlarmResetPB AND #EnableAlarm,   // TOF
                 PT := T#30S,
                 ET => "NotUsedTime");
   #AlarmOB80 := #TimerOffOB80.Q;
END_REGION

REGION Network 25: **** 2.2 - Alarms - Alarm Generation **** Alarm exception OB81
   // Alarm exception OB81
   #TimerOffOB81(IN := ("CPUOB81Execution" <> #MemOB81Execution) AND NOT #I_AlarmResetPB AND #EnableAlarm,   // TOF
                 PT := T#30S,
                 ET => "NotUsedTime");
   #AlarmOB81 := #TimerOffOB81.Q;
END_REGION

REGION Network 26: **** 2.2 - Alarms - Alarm Generation **** Alarm exception OB82
   // Alarm exception OB82
   #AlarmOB82 := "FALSE";
END_REGION

REGION Network 27: **** 2.2 - Alarms - Alarm Generation **** Alarm exception OB83
   // Alarm exception OB83
   #TimerOffB83(IN := ("CPUOB83Execution" <> #MemOB83Execution) AND NOT #I_AlarmResetPB AND #EnableAlarm,   // TOF
                PT := T#30S,
                ET => "NotUsedTime");
   #AlarmOB83 := #TimerOffB83.Q;
END_REGION

REGION Network 28: **** 2.2 - Alarms - Alarm Generation **** Alarm exception OB84
   // Alarm exception OB84
   #TimerOffOB84(IN := ("CPUOB84Execution" <> #MemOB84Execution) AND NOT #I_AlarmResetPB AND #EnableAlarm,   // TOF
                 PT := T#30S,
                 ET => "NotUsedTime");
   #AlarmOB84 := #TimerOffOB84.Q;
END_REGION

REGION Network 29: **** 2.2 - Alarms - Alarm Generation **** Alarm exception OB85
   // Alarm exception OB85
   #TimerOffOB85(IN := ("CPUOB85Execution" <> #MemOB85Execution) AND NOT #I_AlarmResetPB AND #EnableAlarm,   // TOF
                 PT := T#30S,
                 ET => "NotUsedTime");
   #AlarmOB85 := #TimerOffOB85.Q;
END_REGION

REGION Network 30: **** 2.2 - Alarms - Alarm Generation **** Alarm exception OB86
   // Alarm exception OB86
   #TimerOffOB86(IN := ("CPUOB86Execution" <> #MemOB86Execution) AND NOT #I_AlarmResetPB AND #EnableAlarm,   // TOF
                 PT := T#30S,
                 ET => "NotUsedTime");
   #AlarmOB86 := #TimerOffOB86.Q;
END_REGION

REGION Network 31: **** 2.2 - Alarms - Alarm Generation **** Alarm exception OB87
   // Alarm exception OB87
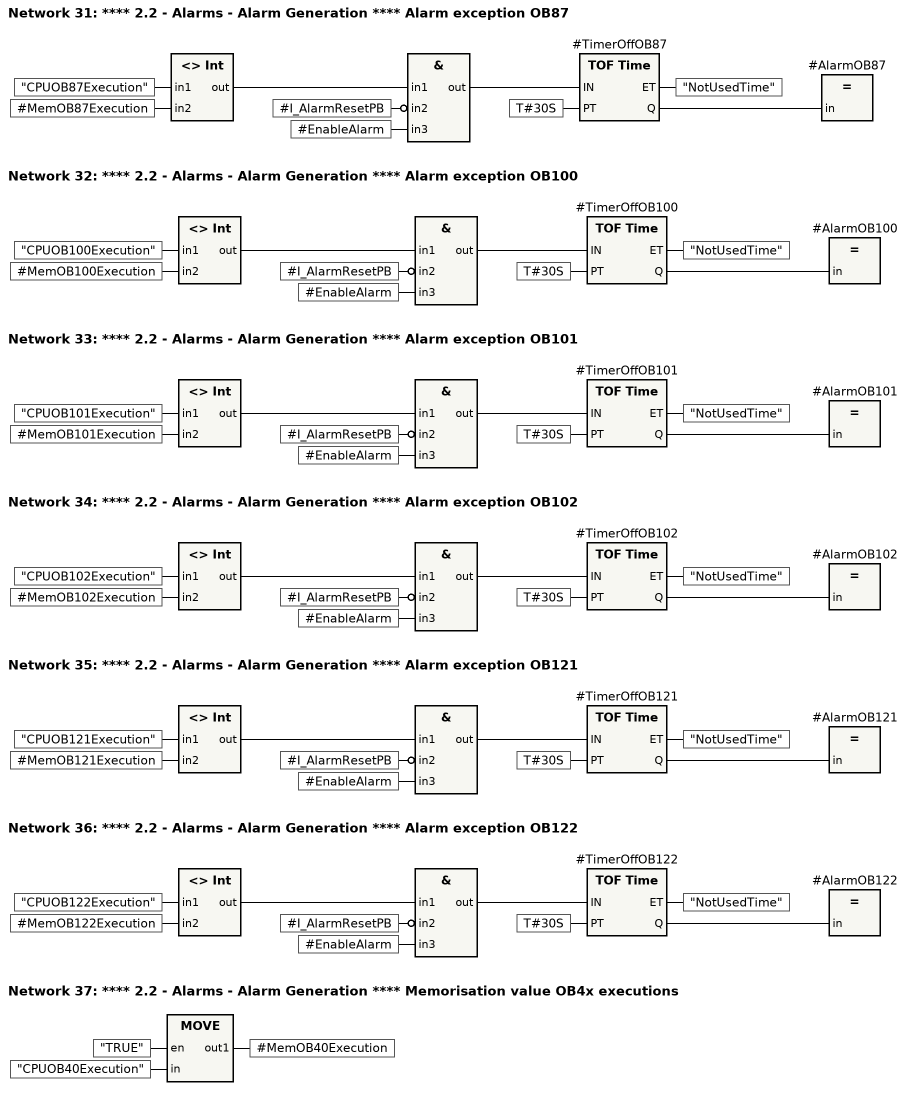
   #TimerOffOB87(IN := ("CPUOB87Execution" <> #MemOB87Execution) AND NOT #I_AlarmResetPB AND #EnableAlarm,   // TOF
                 PT := T#30S,
                 ET => "NotUsedTime");
   #AlarmOB87 := #TimerOffOB87.Q;
END_REGION

REGION Network 32: **** 2.2 - Alarms - Alarm Generation **** Alarm exception OB100
   // Alarm exception OB100
   #TimerOffOB100(IN := ("CPUOB100Execution" <> #MemOB100Execution) AND NOT #I_AlarmResetPB AND #EnableAlarm,   // TOF
                  PT := T#30S,
                  ET => "NotUsedTime");
   #AlarmOB100 := #TimerOffOB100.Q;
END_REGION

REGION Network 33: **** 2.2 - Alarms - Alarm Generation **** Alarm exception OB101
   // Alarm exception OB101
   #TimerOffOB101(IN := ("CPUOB101Execution" <> #MemOB101Execution) AND NOT #I_AlarmResetPB AND #EnableAlarm,   // TOF
                  PT := T#30S,
                  ET => "NotUsedTime");
   #AlarmOB101 := #TimerOffOB101.Q;
END_REGION

REGION Network 34: **** 2.2 - Alarms - Alarm Generation **** Alarm exception OB102
   // Alarm exception OB102
   #TimerOffOB102(IN := ("CPUOB102Execution" <> #MemOB102Execution) AND NOT #I_AlarmResetPB AND #EnableAlarm,   // TOF
                  PT := T#30S,
                  ET => "NotUsedTime");
   #AlarmOB102 := #TimerOffOB102.Q;
END_REGION

REGION Network 35: **** 2.2 - Alarms - Alarm Generation **** Alarm exception OB121
   // Alarm exception OB121
   #TimerOffOB121(IN := ("CPUOB121Execution" <> #MemOB121Execution) AND NOT #I_AlarmResetPB AND #EnableAlarm,   // TOF
                  PT := T#30S,
                  ET => "NotUsedTime");
   #AlarmOB121 := #TimerOffOB121.Q;
END_REGION

REGION Network 36: **** 2.2 - Alarms - Alarm Generation **** Alarm exception OB122
   // Alarm exception OB122
   #TimerOffOB122(IN := ("CPUOB122Execution" <> #MemOB122Execution) AND NOT #I_AlarmResetPB AND #EnableAlarm,   // TOF
                  PT := T#30S,
                  ET => "NotUsedTime");
   #AlarmOB122 := #TimerOffOB122.Q;
END_REGION

REGION Network 37: **** 2.2 - Alarms - Alarm Generation **** Memorisation value OB4x executions
   // Memorisation value OB4x executions
   IF "TRUE" THEN #MemOB40Execution := "CPUOB40Execution"; END_IF;
END_REGION

REGION Network 38: **** 2.2 - Alarms - Alarm Generation **** Memorisation value OB8x executions
   // Memorisation value OB8x executions
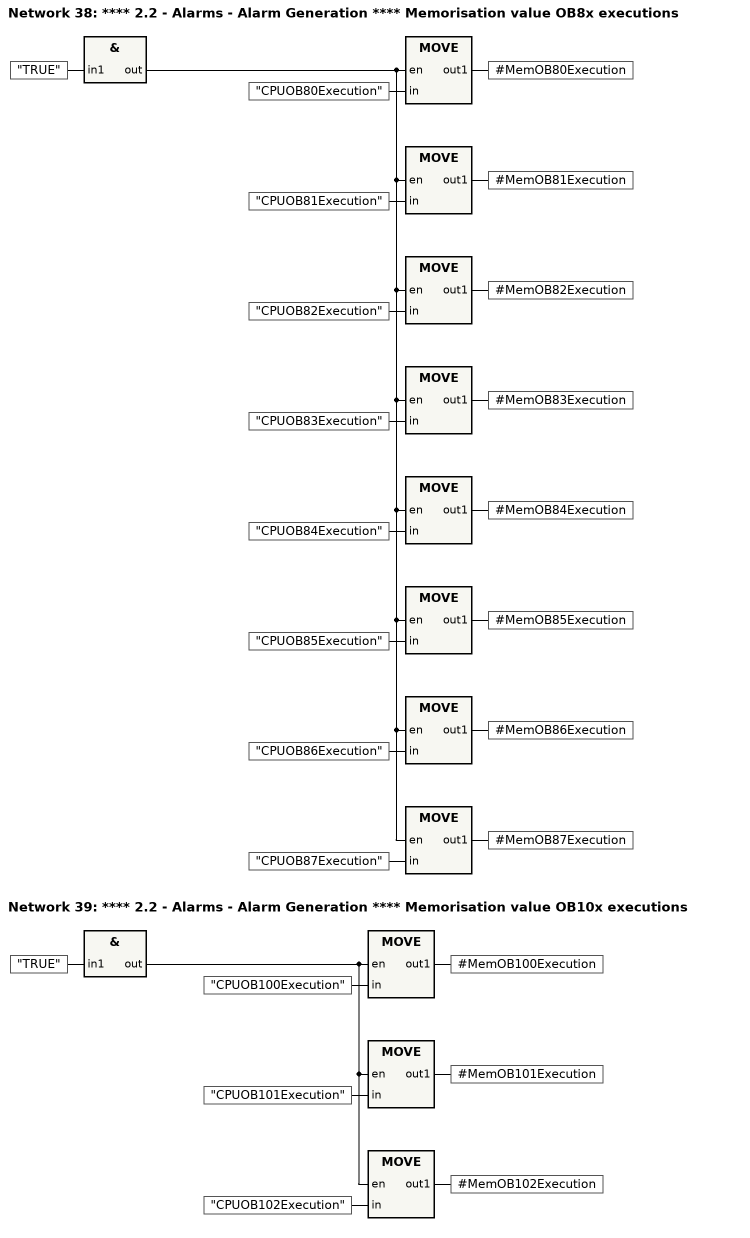
   IF "TRUE" THEN
       #MemOB80Execution := "CPUOB80Execution";
       #MemOB81Execution := "CPUOB81Execution";
       #MemOB82Execution := "CPUOB82Execution";
       #MemOB83Execution := "CPUOB83Execution";
       #MemOB84Execution := "CPUOB84Execution";
       #MemOB85Execution := "CPUOB85Execution";
       #MemOB86Execution := "CPUOB86Execution";
       #MemOB87Execution := "CPUOB87Execution";
   END_IF;
END_REGION

REGION Network 39: **** 2.2 - Alarms - Alarm Generation **** Memorisation value OB10x executions
   // Memorisation value OB10x executions
   IF "TRUE" THEN
       #MemOB100Execution := "CPUOB100Execution";
       #MemOB101Execution := "CPUOB101Execution";
       #MemOB102Execution := "CPUOB102Execution";
   END_IF;
END_REGION

REGION Network 40: **** 2.2 - Alarms - Alarm Generation **** Memorisation value OB12x executions
   // Memorisation value OB12x executions
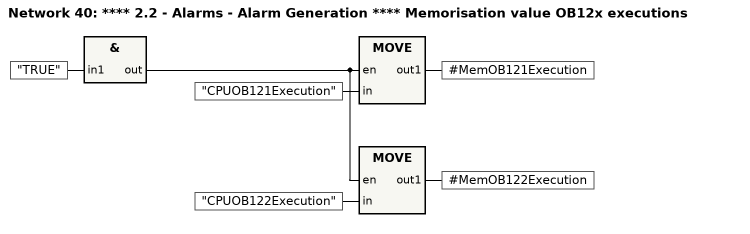
   IF "TRUE" THEN
       #MemOB121Execution := "CPUOB121Execution";
       #MemOB122Execution := "CPUOB122Execution";
   END_IF;
END_REGION

REGION Network 41: **** 2.2 - Alarms - Alarm Generation **** Alarms exception OB40,80,81,82,83,84,85,86,87,100
   // Alarms exception OB40,80,81,82,83,84,85,86,87,100
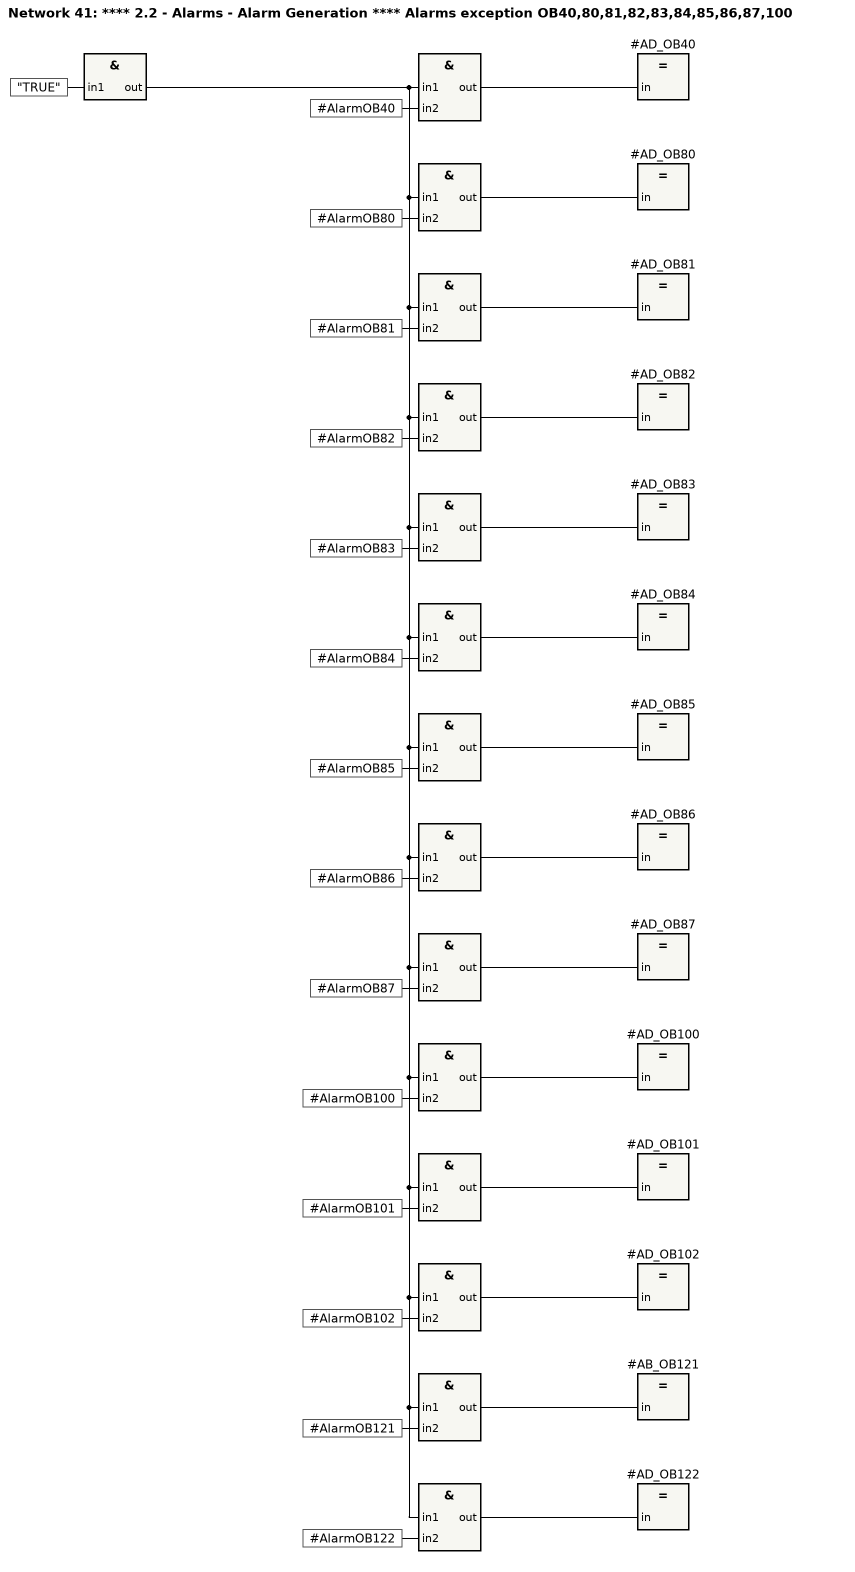
   #AD_OB40 := "TRUE" AND #AlarmOB40;
   #AD_OB80 := "TRUE" AND #AlarmOB80;
   #AD_OB81 := "TRUE" AND #AlarmOB81;
   #AD_OB82 := "TRUE" AND #AlarmOB82;
   #AD_OB83 := "TRUE" AND #AlarmOB83;
   #AD_OB84 := "TRUE" AND #AlarmOB84;
   #AD_OB85 := "TRUE" AND #AlarmOB85;
   #AD_OB86 := "TRUE" AND #AlarmOB86;
   #AD_OB87 := "TRUE" AND #AlarmOB87;
   #AD_OB100 := "TRUE" AND #AlarmOB100;
   #AD_OB101 := "TRUE" AND #AlarmOB101;
   #AD_OB102 := "TRUE" AND #AlarmOB102;
   #AB_OB121 := "TRUE" AND #AlarmOB121;
   #AD_OB122 := "TRUE" AND #AlarmOB122;
END_REGION

REGION Network 42: **** 2.2 - Alarms - Alarm Generation **** Calibration MovUnits / **** 2.2 - Alarms - Alarm Generation **** Info -> Redo Overtime calibration MovUnit
   // Alarms exception OB40,80,81,82,83,84,85,86,87,100 / Calibration MovUnits
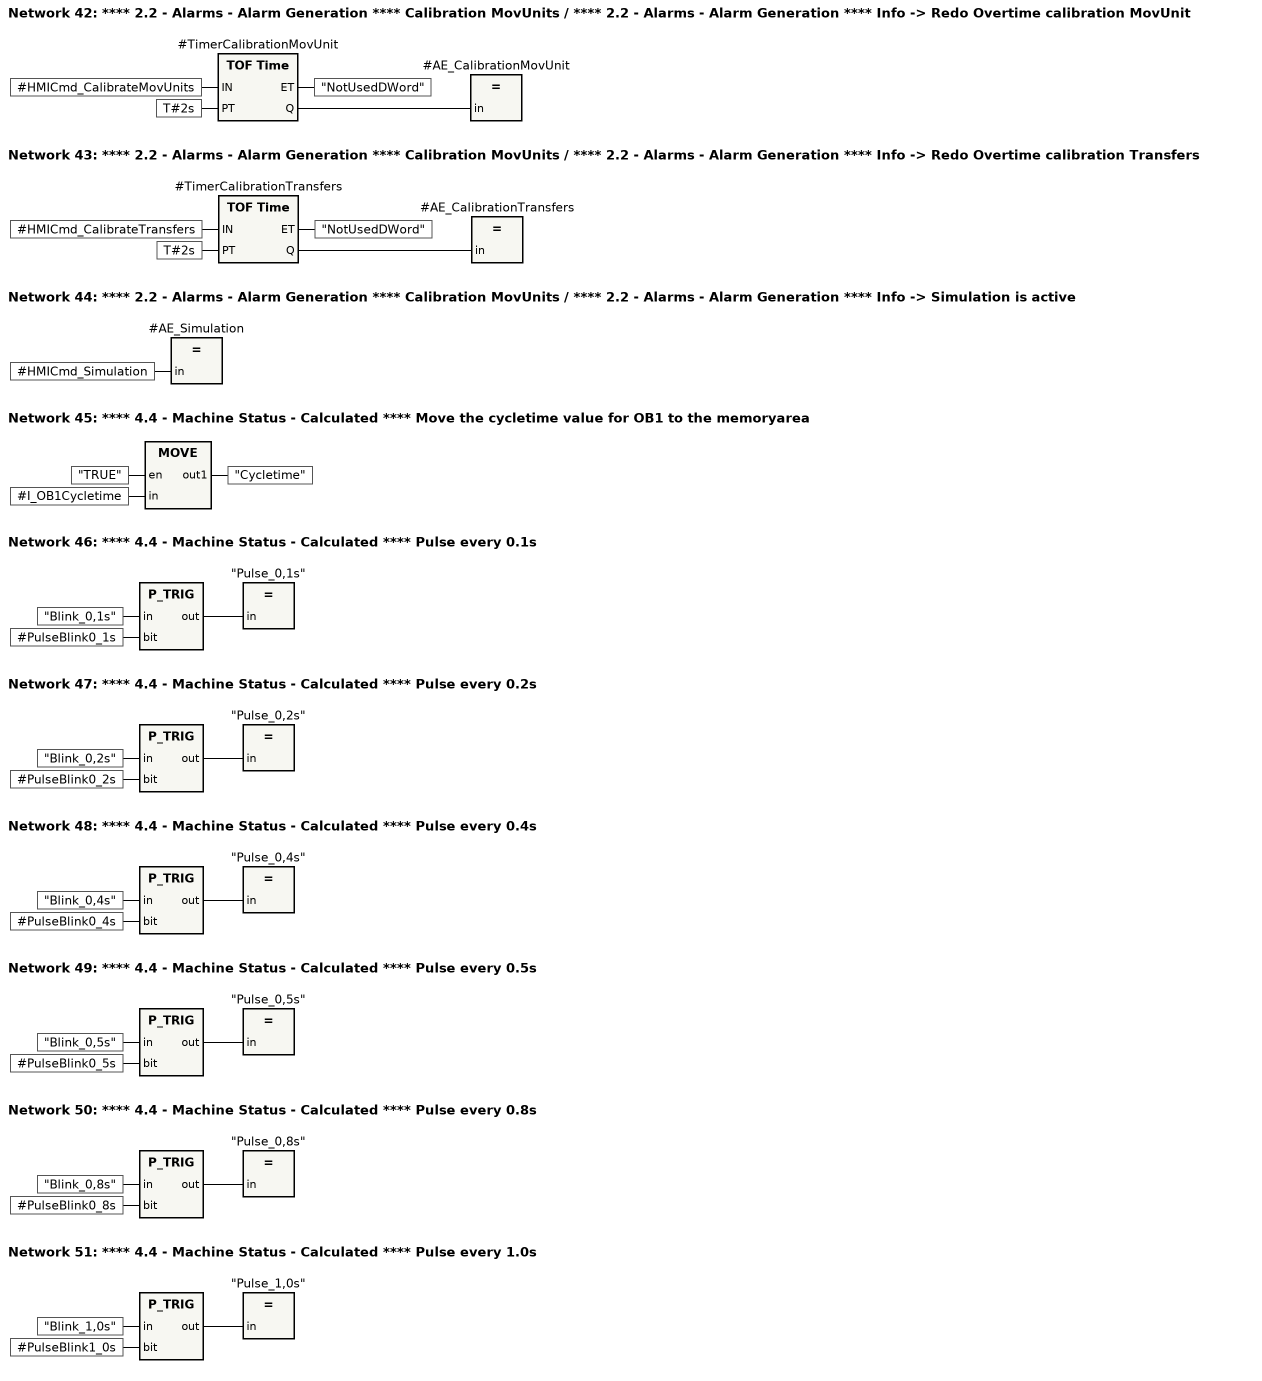
   #TimerCalibrationMovUnit(IN := #HMICmd_CalibrateMovUnits, PT := T#2s, ET => "NotUsedDWord");   // TOF
   #AE_CalibrationMovUnit := #TimerCalibrationMovUnit.Q;
END_REGION

REGION Network 43: **** 2.2 - Alarms - Alarm Generation **** Calibration MovUnits / **** 2.2 - Alarms - Alarm Generation **** Info -> Redo Overtime calibration Transfers
   // Alarms exception OB40,80,81,82,83,84,85,86,87,100 / Calibration MovUnits
   #TimerCalibrationTransfers(IN := #HMICmd_CalibrateTransfers, PT := T#2s, ET => "NotUsedDWord");   // TOF
   #AE_CalibrationTransfers := #TimerCalibrationTransfers.Q;
END_REGION

REGION Network 44: **** 2.2 - Alarms - Alarm Generation **** Calibration MovUnits / **** 2.2 - Alarms - Alarm Generation **** Info -> Simulation is active
   // Alarms exception OB40,80,81,82,83,84,85,86,87,100 / Calibration MovUnits
   #AE_Simulation := #HMICmd_Simulation;
END_REGION

REGION Network 45: **** 4.4 - Machine Status - Calculated **** Move the cycletime value for OB1 to the memoryarea
   // Move the cycletime value for OB1 to the memory area
   IF "TRUE" THEN "Cycletime" := #I_OB1Cycletime; END_IF;
END_REGION

REGION Network 46: **** 4.4 - Machine Status - Calculated **** Pulse every 0.1s
   // Pulse every 0.1s
   #_w1 := "Blink_0,1s" AND NOT #PulseBlink0_1s;   // rising edge
   #PulseBlink0_1s := "Blink_0,1s";
   "Pulse_0,1s" := #_w1;
END_REGION

REGION Network 47: **** 4.4 - Machine Status - Calculated **** Pulse every 0.2s
   // Pulse every 0.2s
   #_w1 := "Blink_0,2s" AND NOT #PulseBlink0_2s;   // rising edge
   #PulseBlink0_2s := "Blink_0,2s";
   "Pulse_0,2s" := #_w1;
END_REGION

REGION Network 48: **** 4.4 - Machine Status - Calculated **** Pulse every 0.4s
   // Pulse every 0.4s
   #_w1 := "Blink_0,4s" AND NOT #PulseBlink0_4s;   // rising edge
   #PulseBlink0_4s := "Blink_0,4s";
   "Pulse_0,4s" := #_w1;
END_REGION

REGION Network 49: **** 4.4 - Machine Status - Calculated **** Pulse every 0.5s
   // Pulse every 0.5s
   #_w1 := "Blink_0,5s" AND NOT #PulseBlink0_5s;   // rising edge
   #PulseBlink0_5s := "Blink_0,5s";
   "Pulse_0,5s" := #_w1;
END_REGION

REGION Network 50: **** 4.4 - Machine Status - Calculated **** Pulse every 0.8s
   // Pulse every 0.8s
   #_w1 := "Blink_0,8s" AND NOT #PulseBlink0_8s;   // rising edge
   #PulseBlink0_8s := "Blink_0,8s";
   "Pulse_0,8s" := #_w1;
END_REGION

REGION Network 51: **** 4.4 - Machine Status - Calculated **** Pulse every 1.0s
   // Pulse every 1.0s
   #_w1 := "Blink_1,0s" AND NOT #PulseBlink1_0s;   // rising edge
   #PulseBlink1_0s := "Blink_1,0s";
   "Pulse_1,0s" := #_w1;
END_REGION

REGION Network 52: **** 4.4 - Machine Status - Calculated **** Pulse every 1.6s
   // Pulse every 1.6s
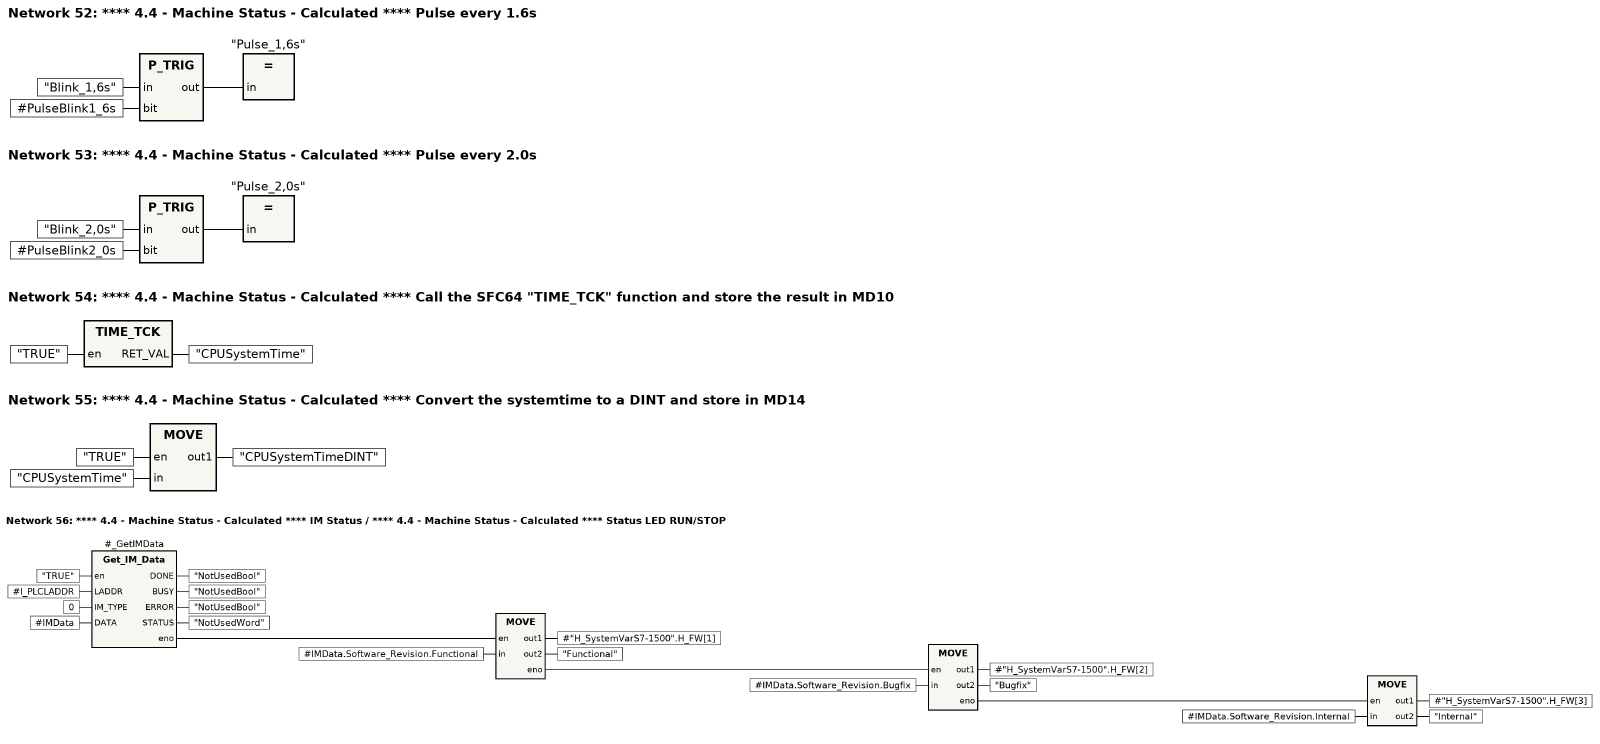
   #_w1 := "Blink_1,6s" AND NOT #PulseBlink1_6s;   // rising edge
   #PulseBlink1_6s := "Blink_1,6s";
   "Pulse_1,6s" := #_w1;
END_REGION

REGION Network 53: **** 4.4 - Machine Status - Calculated **** Pulse every 2.0s
   // Pulse every 2.0s
   #_w1 := "Blink_2,0s" AND NOT #PulseBlink2_0s;   // rising edge
   #PulseBlink2_0s := "Blink_2,0s";
   "Pulse_2,0s" := #_w1;
END_REGION

REGION Network 54: **** 4.4 - Machine Status - Calculated **** Call the SFC64 "TIME_TCK" function and store the result in MD10
   // Call the SFC64 "TIME_TCK" function and store the result in MD10
   IF "TRUE" THEN "CPUSystemTime" := TIME_TCK(); END_IF;
END_REGION

REGION Network 55: **** 4.4 - Machine Status - Calculated **** Convert the systemtime to a DINT and store in MD14
   // Convert the systemtime to a DINT and store in MD14
   IF "TRUE" THEN "CPUSystemTimeDINT" := "CPUSystemTime"; END_IF;
END_REGION

REGION Network 56: **** 4.4 - Machine Status - Calculated **** IM Status / **** 4.4 - Machine Status - Calculated **** Status LED RUN/STOP
   // IM Status
   // Status LEDs
   // LED1 SF :  Group error
   #_GetIMData(EN := "TRUE",   // Get_IM_Data
               LADDR := #I_PLCLADDR,
               IM_TYPE := 0,
               DATA := #IMData,
               DONE => "NotUsedBool",
               BUSY => "NotUsedBool",
               ERROR => "NotUsedBool",
               STATUS => "NotUsedWord",
               ENO => #_w1);
   IF #_w1 THEN
       #"H_SystemVarS7-1500".H_FW[1] := #IMData.Software_Revision.Functional;
       "Functional" := #IMData.Software_Revision.Functional;
       #"H_SystemVarS7-1500".H_FW[2] := #IMData.Software_Revision.Bugfix;
       "Bugfix" := #IMData.Software_Revision.Bugfix;
       #"H_SystemVarS7-1500".H_FW[3] := #IMData.Software_Revision.Internal;
       "Internal" := #IMData.Software_Revision.Internal;
   END_IF;
END_REGION

REGION Network 57: **** 4.4 - Machine Status - Calculated **** Status LED RUN/STOP
   // Status LEDs
   // LED1 SF :  Group error
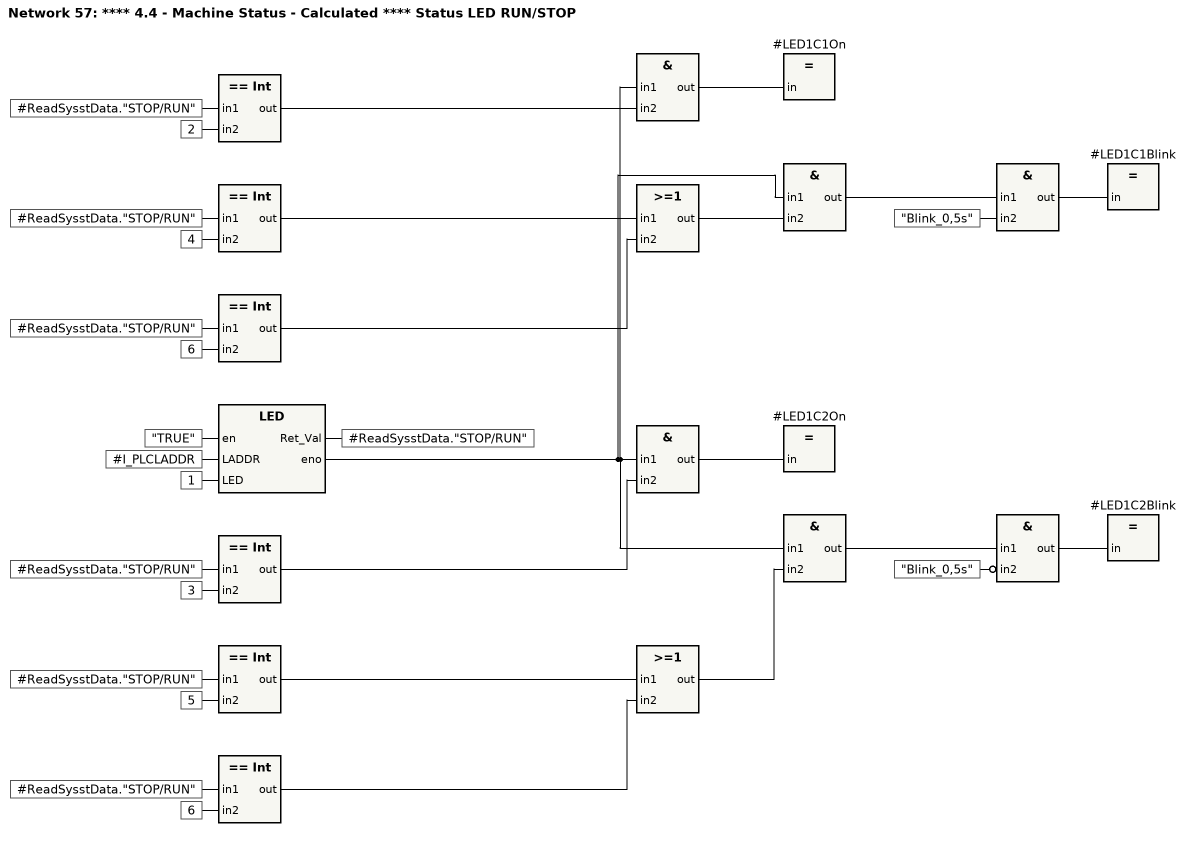
   #ReadSysstData."STOP/RUN" := LED(EN := "TRUE", LADDR := #I_PLCLADDR, LED := 1, ENO => #_w1);
   #LED1C1On := #_w1 AND (#ReadSysstData."STOP/RUN" = 2);
   #LED1C2On := #_w1 AND (#ReadSysstData."STOP/RUN" = 3);
   #LED1C1Blink := #_w1 AND ((#ReadSysstData."STOP/RUN" = 4) OR (#ReadSysstData."STOP/RUN" = 6)) AND "Blink_0,5s";
   #LED1C2Blink := #_w1 AND ((#ReadSysstData."STOP/RUN" = 5) OR (#ReadSysstData."STOP/RUN" = 6)) AND NOT "Blink_0,5s";
END_REGION

REGION Network 58: **** 4.4 - Machine Status - Calculated **** Status LED ERROR
   // Status LEDs
   // LED4 RUN
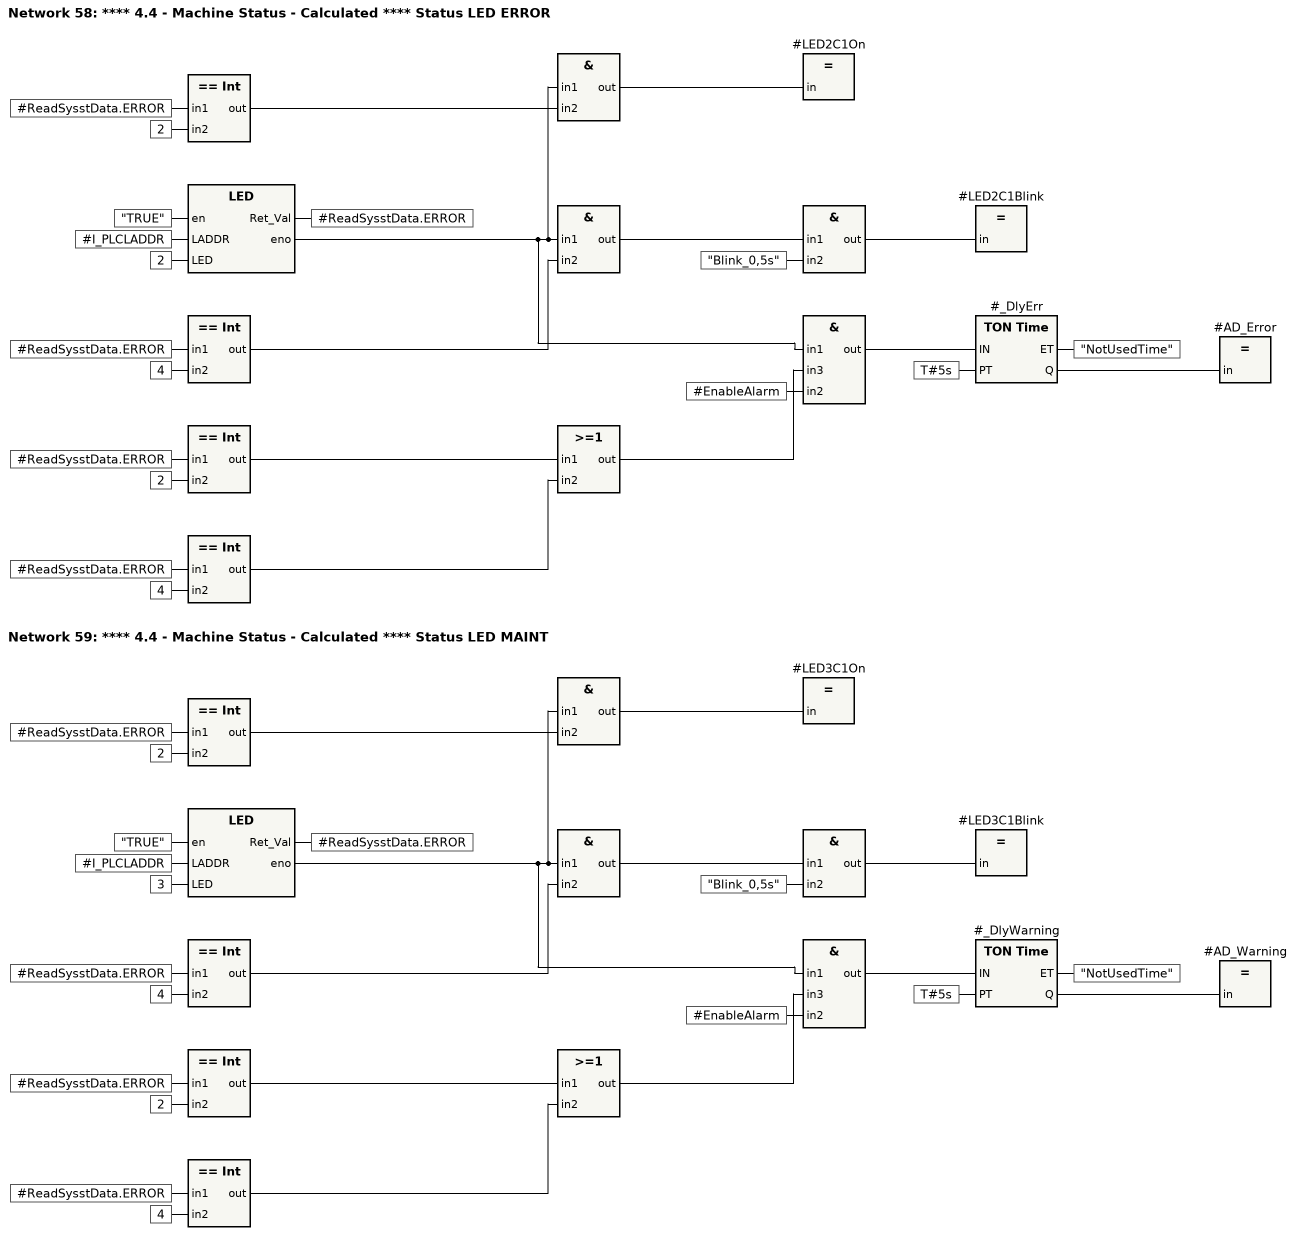
   #ReadSysstData.ERROR := LED(EN := "TRUE", LADDR := #I_PLCLADDR, LED := 2, ENO => #_w1);
   #LED2C1On := #_w1 AND (#ReadSysstData.ERROR = 2);
   #LED2C1Blink := #_w1 AND (#ReadSysstData.ERROR = 4) AND "Blink_0,5s";
   #_DlyErr(IN := #_w1 AND ((#ReadSysstData.ERROR = 2) OR (#ReadSysstData.ERROR = 4)) AND #EnableAlarm,   // TON
            PT := T#5s,
            ET => "NotUsedTime");
   #AD_Error := #_DlyErr.Q;
END_REGION

REGION Network 59: **** 4.4 - Machine Status - Calculated **** Status LED MAINT
   // Status LEDs
   // LED5 STOP
   #ReadSysstData.ERROR := LED(EN := "TRUE", LADDR := #I_PLCLADDR, LED := 3, ENO => #_w1);
   #LED3C1On := #_w1 AND (#ReadSysstData.ERROR = 2);
   #LED3C1Blink := #_w1 AND (#ReadSysstData.ERROR = 4) AND "Blink_0,5s";
   #_DlyWarning(IN := #_w1 AND ((#ReadSysstData.ERROR = 2) OR (#ReadSysstData.ERROR = 4)) AND #EnableAlarm,   // TON
                PT := T#5s,
                ET => "NotUsedTime");
   #AD_Warning := #_DlyWarning.Q;
END_REGION

REGION Network 60: **** 4.4 - Machine Status - Calculated **** Read SystemTime
   // Read SystemTime
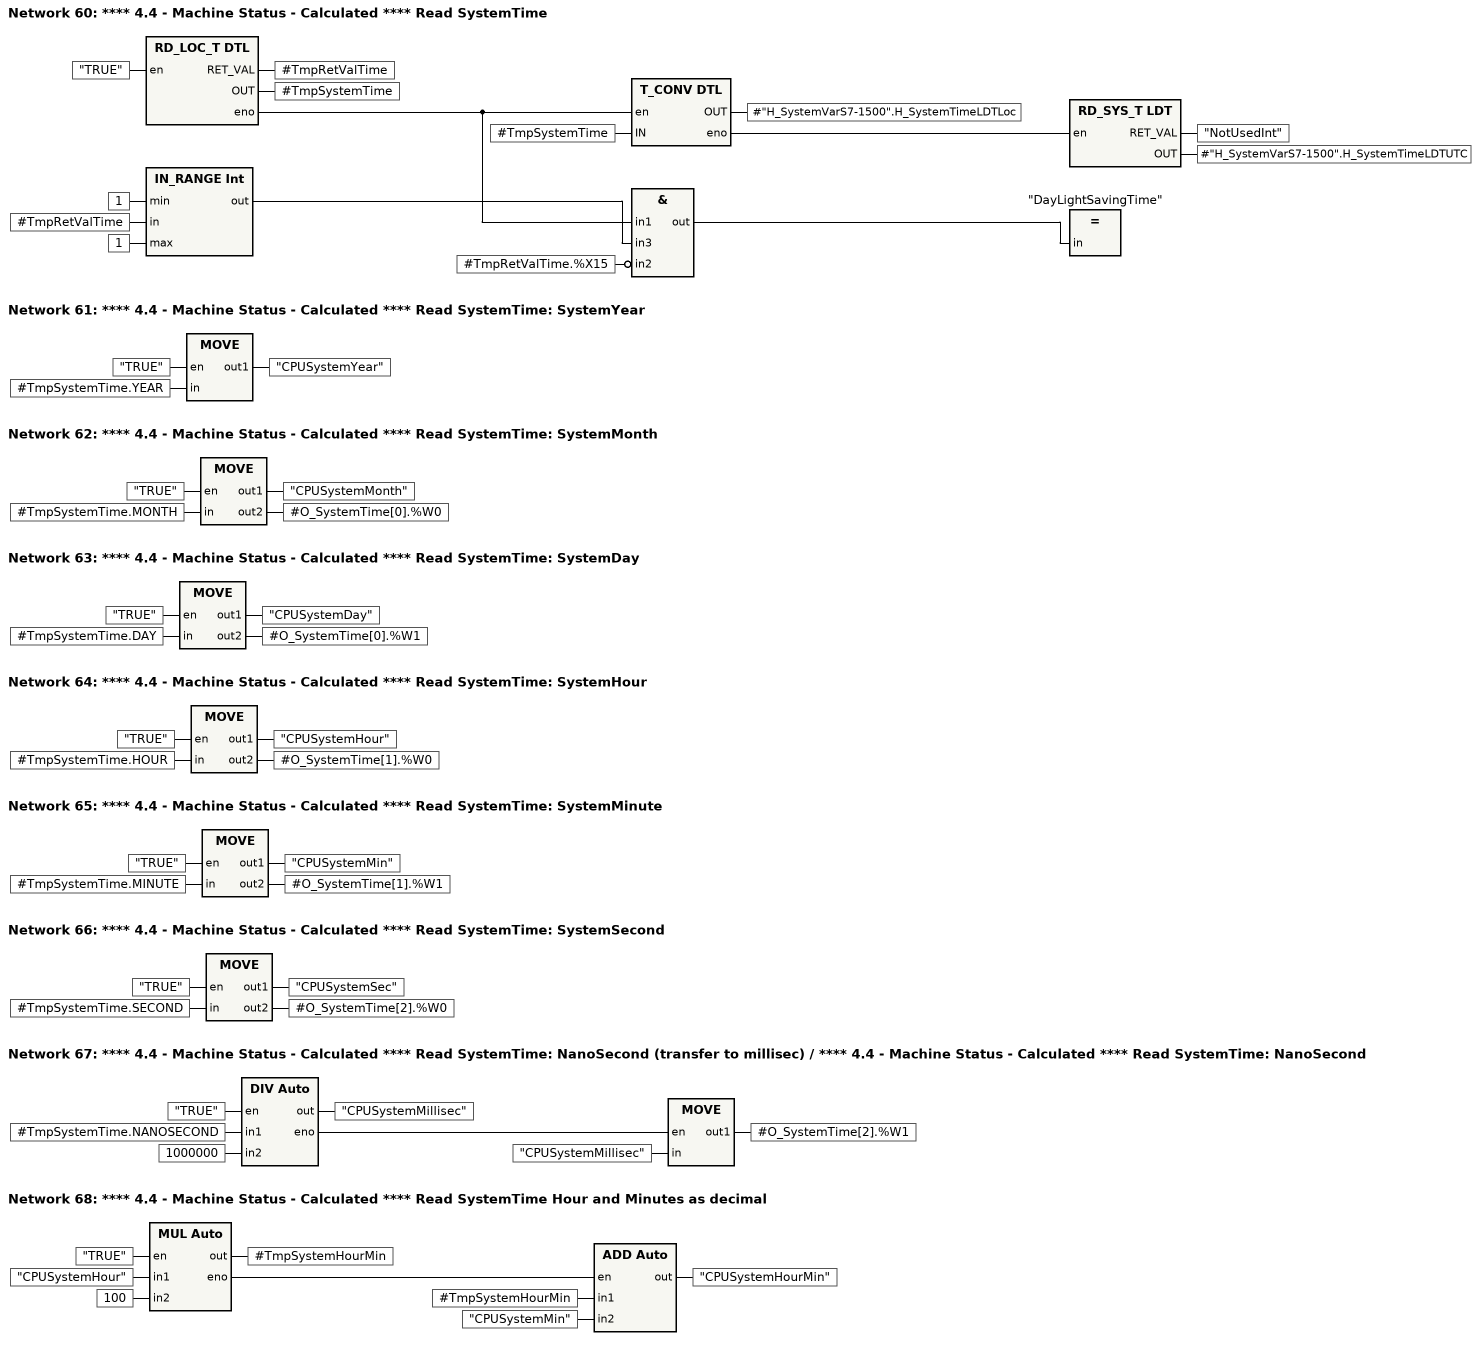
   #TmpRetValTime := RD_LOC_T(EN := "TRUE", OUT => #TmpSystemTime, ENO => #_w1);
   T_CONV(EN := #_w1, IN := #TmpSystemTime, OUT => #"H_SystemVarS7-1500".H_SystemTimeLDTLoc, ENO => #_w2);
   IF #_w2 THEN "NotUsedInt" := RD_SYS_T(OUT => #"H_SystemVarS7-1500".H_SystemTimeLDTUTC); END_IF;
   "DayLightSavingTime" := #_w1 AND (1 <= #TmpRetValTime) AND (#TmpRetValTime <= 1) AND NOT #TmpRetValTime.%X15;
END_REGION

REGION Network 61: **** 4.4 - Machine Status - Calculated **** Read SystemTime: SystemYear
   // Read SystemTime: SystemYear
   IF "TRUE" THEN "CPUSystemYear" := #TmpSystemTime.YEAR; END_IF;
END_REGION

REGION Network 62: **** 4.4 - Machine Status - Calculated **** Read SystemTime: SystemMonth
   // Read SystemTime: SystemMonth
   IF "TRUE" THEN
       "CPUSystemMonth" := #TmpSystemTime.MONTH;
       #O_SystemTime[0].%W0 := #TmpSystemTime.MONTH;
   END_IF;
END_REGION

REGION Network 63: **** 4.4 - Machine Status - Calculated **** Read SystemTime: SystemDay
   // Read SystemTime: SystemDay
   IF "TRUE" THEN
       "CPUSystemDay" := #TmpSystemTime.DAY;
       #O_SystemTime[0].%W1 := #TmpSystemTime.DAY;
   END_IF;
END_REGION

REGION Network 64: **** 4.4 - Machine Status - Calculated **** Read SystemTime: SystemHour
   // Read SystemTime: SystemHour
   IF "TRUE" THEN
       "CPUSystemHour" := #TmpSystemTime.HOUR;
       #O_SystemTime[1].%W0 := #TmpSystemTime.HOUR;
   END_IF;
END_REGION

REGION Network 65: **** 4.4 - Machine Status - Calculated **** Read SystemTime: SystemMinute
   // Read SystemTime: SystemMinute
   IF "TRUE" THEN
       "CPUSystemMin" := #TmpSystemTime.MINUTE;
       #O_SystemTime[1].%W1 := #TmpSystemTime.MINUTE;
   END_IF;
END_REGION

REGION Network 66: **** 4.4 - Machine Status - Calculated **** Read SystemTime: SystemSecond
   // Read SystemTime: SystemSecond
   IF "TRUE" THEN
       "CPUSystemSec" := #TmpSystemTime.SECOND;
       #O_SystemTime[2].%W0 := #TmpSystemTime.SECOND;
   END_IF;
END_REGION

REGION Network 67: **** 4.4 - Machine Status - Calculated **** Read SystemTime: NanoSecond (transfer to millisec) / **** 4.4 - Machine Status - Calculated **** Read SystemTime: NanoSecond
   // Read SystemTime: NanoSecond (transfer to millisec) / Read SystemTime: NanoSecond
   IF "TRUE" THEN
       "CPUSystemMillisec" := #TmpSystemTime.NANOSECOND / 1000000;
       #O_SystemTime[2].%W1 := "CPUSystemMillisec";
   END_IF;
END_REGION

REGION Network 68: **** 4.4 - Machine Status - Calculated **** Read SystemTime Hour and Minutes as decimal
   // Makes an integer holding the combined values of hour and minute in the format 
   // hh:mm. This is used to compare the clock with time values from the 
   // steering bridge. (ex. if the value is 2312 it represents the time 
   // 23:12 and the value 32 represents 00:32)
   IF "TRUE" THEN
       #TmpSystemHourMin := "CPUSystemHour" * 100;
       "CPUSystemHourMin" := #TmpSystemHourMin + "CPUSystemMin";
   END_IF;
END_REGION

REGION Network 69: **** 4.4 - Machine Status - Calculated **** Move the SystemWeekDay to a temporary variable / **** 4.4 - Machine Status - Calculated **** Move the weekday to a temporary variable
   // Move the SystemWeekDay to a temporary variable / Move the weekday to a temporary variable
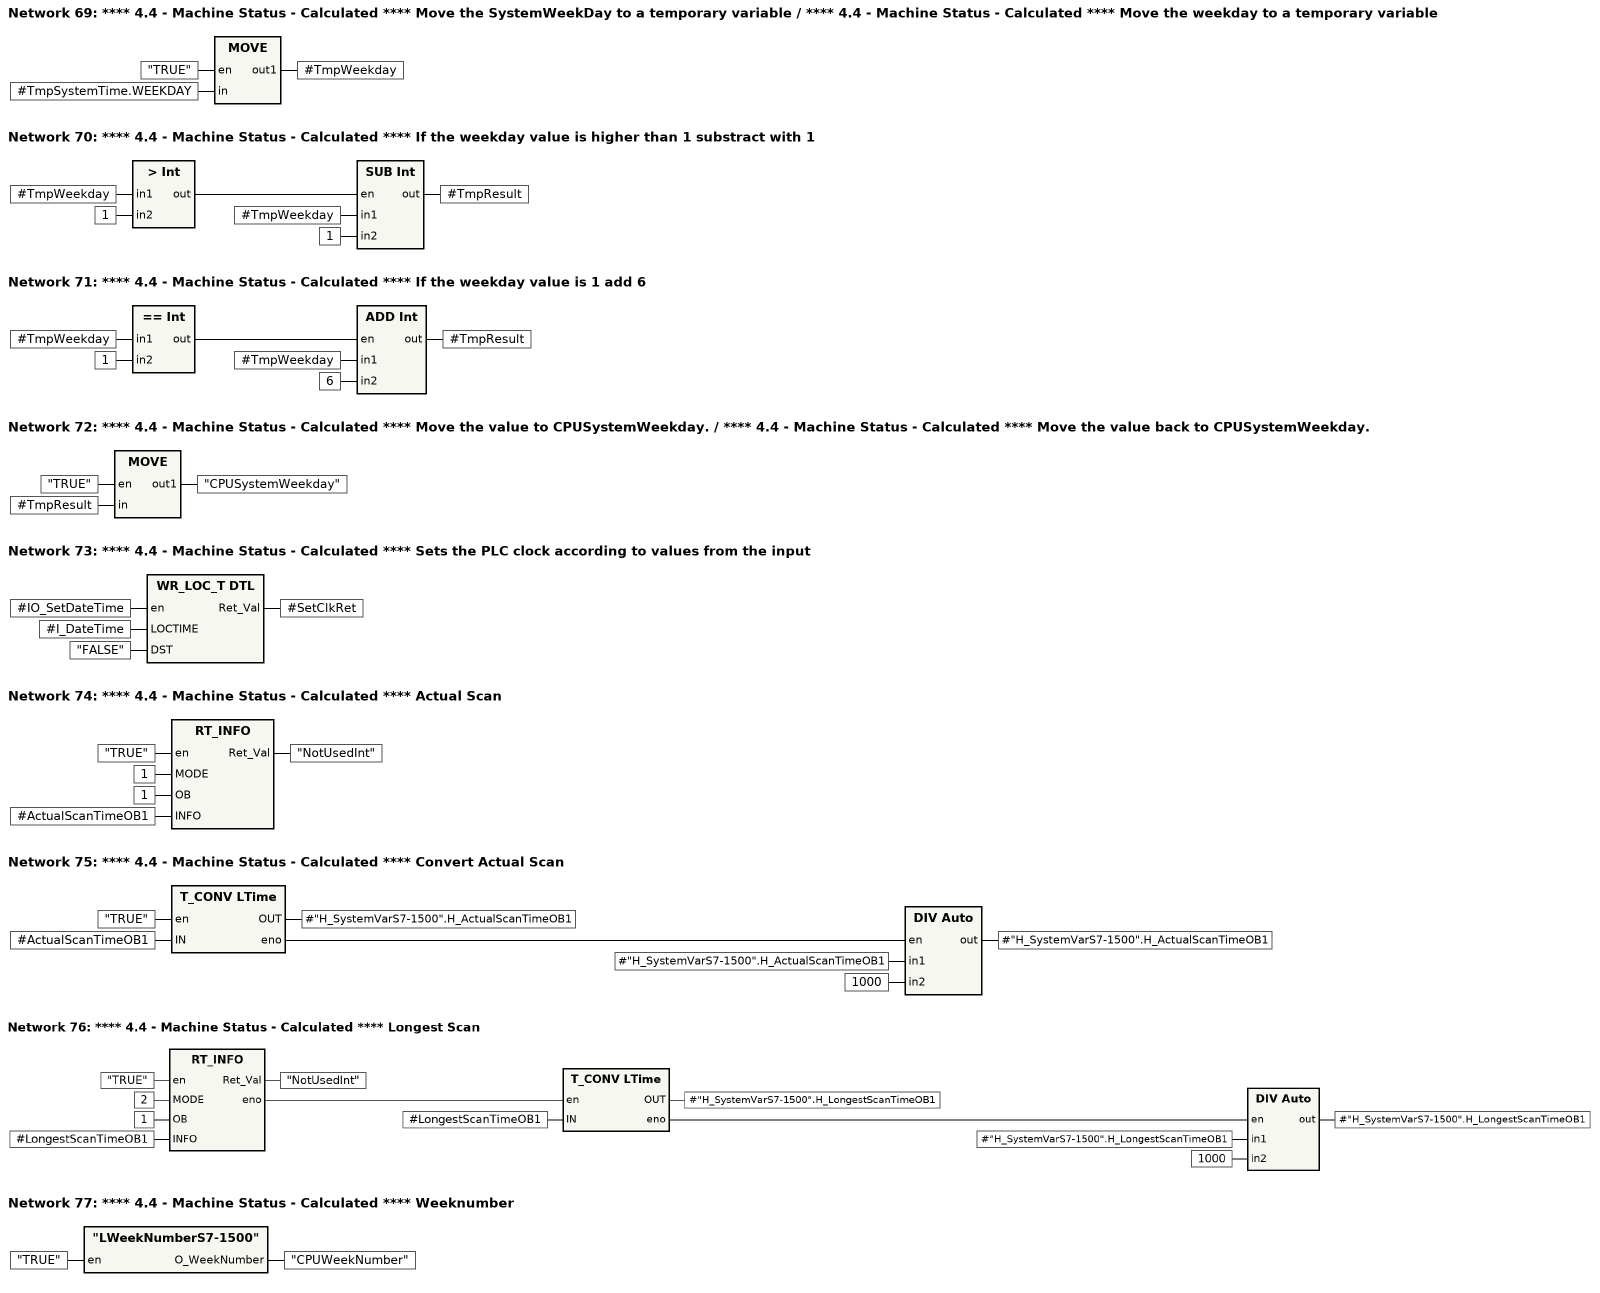
   IF "TRUE" THEN #TmpWeekday := #TmpSystemTime.WEEKDAY; END_IF;
END_REGION

REGION Network 70: **** 4.4 - Machine Status - Calculated **** If the weekday value is higher than 1 substract with 1
   // If the weekday value is higher than 1 substract with 1
   IF #TmpWeekday > 1 THEN #TmpResult := #TmpWeekday - 1; END_IF;
END_REGION

REGION Network 71: **** 4.4 - Machine Status - Calculated **** If the weekday value is 1 add 6
   // If the weekday value is 1 add 6
   IF #TmpWeekday = 1 THEN #TmpResult := #TmpWeekday + 6; END_IF;
END_REGION

REGION Network 72: **** 4.4 - Machine Status - Calculated **** Move the value to CPUSystemWeekday. / **** 4.4 - Machine Status - Calculated **** Move the value back to CPUSystemWeekday.
   // Move the value to CPUSystemWeekday.
   // 1 = Monday
   // 2 = Tuesday
   // 3 = Wednesday
   // 4 = Thursday
   // 5 = Friday
   // 6 = Saturday
   // 7 = Sunday
   // Move the value back to CPUSystemWeekday.
   // 1 = Monday
   // 2 = Tuesday
   // 3 = Wednesday
   // 4 = Thursday
   // 5 = Friday
   // 6 = Saturday
   // 7 = Sunday
   IF "TRUE" THEN "CPUSystemWeekday" := #TmpResult; END_IF;
END_REGION

REGION Network 73: **** 4.4 - Machine Status - Calculated **** Sets the PLC clock according to values from the input
   // Sets the PLC clock according to values from the input
   IF #IO_SetDateTime THEN #SetClkRet := WR_LOC_T(LOCTIME := #I_DateTime, DST := "FALSE"); END_IF;
END_REGION

REGION Network 74: **** 4.4 - Machine Status - Calculated **** Actual Scan
   // Actual Scan
   IF "TRUE" THEN "NotUsedInt" := RT_INFO(MODE := 1, OB := 1, INFO := #ActualScanTimeOB1); END_IF;
END_REGION

REGION Network 75: **** 4.4 - Machine Status - Calculated **** Convert Actual Scan
   // Convert Actual Scan
   T_CONV(EN := "TRUE", IN := #ActualScanTimeOB1, OUT => #"H_SystemVarS7-1500".H_ActualScanTimeOB1, ENO => #_w1);
   IF #_w1 THEN
       #"H_SystemVarS7-1500".H_ActualScanTimeOB1 := #"H_SystemVarS7-1500".H_ActualScanTimeOB1 / 1000;
   END_IF;
END_REGION

REGION Network 76: **** 4.4 - Machine Status - Calculated **** Longest Scan
   // Longest Scan
   "NotUsedInt" := RT_INFO(EN := "TRUE", MODE := 2, OB := 1, INFO := #LongestScanTimeOB1, ENO => #_w1);
   T_CONV(EN := #_w1, IN := #LongestScanTimeOB1, OUT => #"H_SystemVarS7-1500".H_LongestScanTimeOB1, ENO => #_w2);
   IF #_w2 THEN
       #"H_SystemVarS7-1500".H_LongestScanTimeOB1 := #"H_SystemVarS7-1500".H_LongestScanTimeOB1 / 1000;
   END_IF;
END_REGION

REGION Network 77: **** 4.4 - Machine Status - Calculated **** Weeknumber
   // Weeknumber
   IF "TRUE" THEN "LWeekNumberS7-1500"(O_WeekNumber => "CPUWeekNumber"); END_IF;
END_REGION

REGION Network 78: **** 4.4 - Machine Status - Calculated **** Language comparison with default / **** 4.4 - Machine Status - Calculated **** Weeknumber
   // Language comparison with default
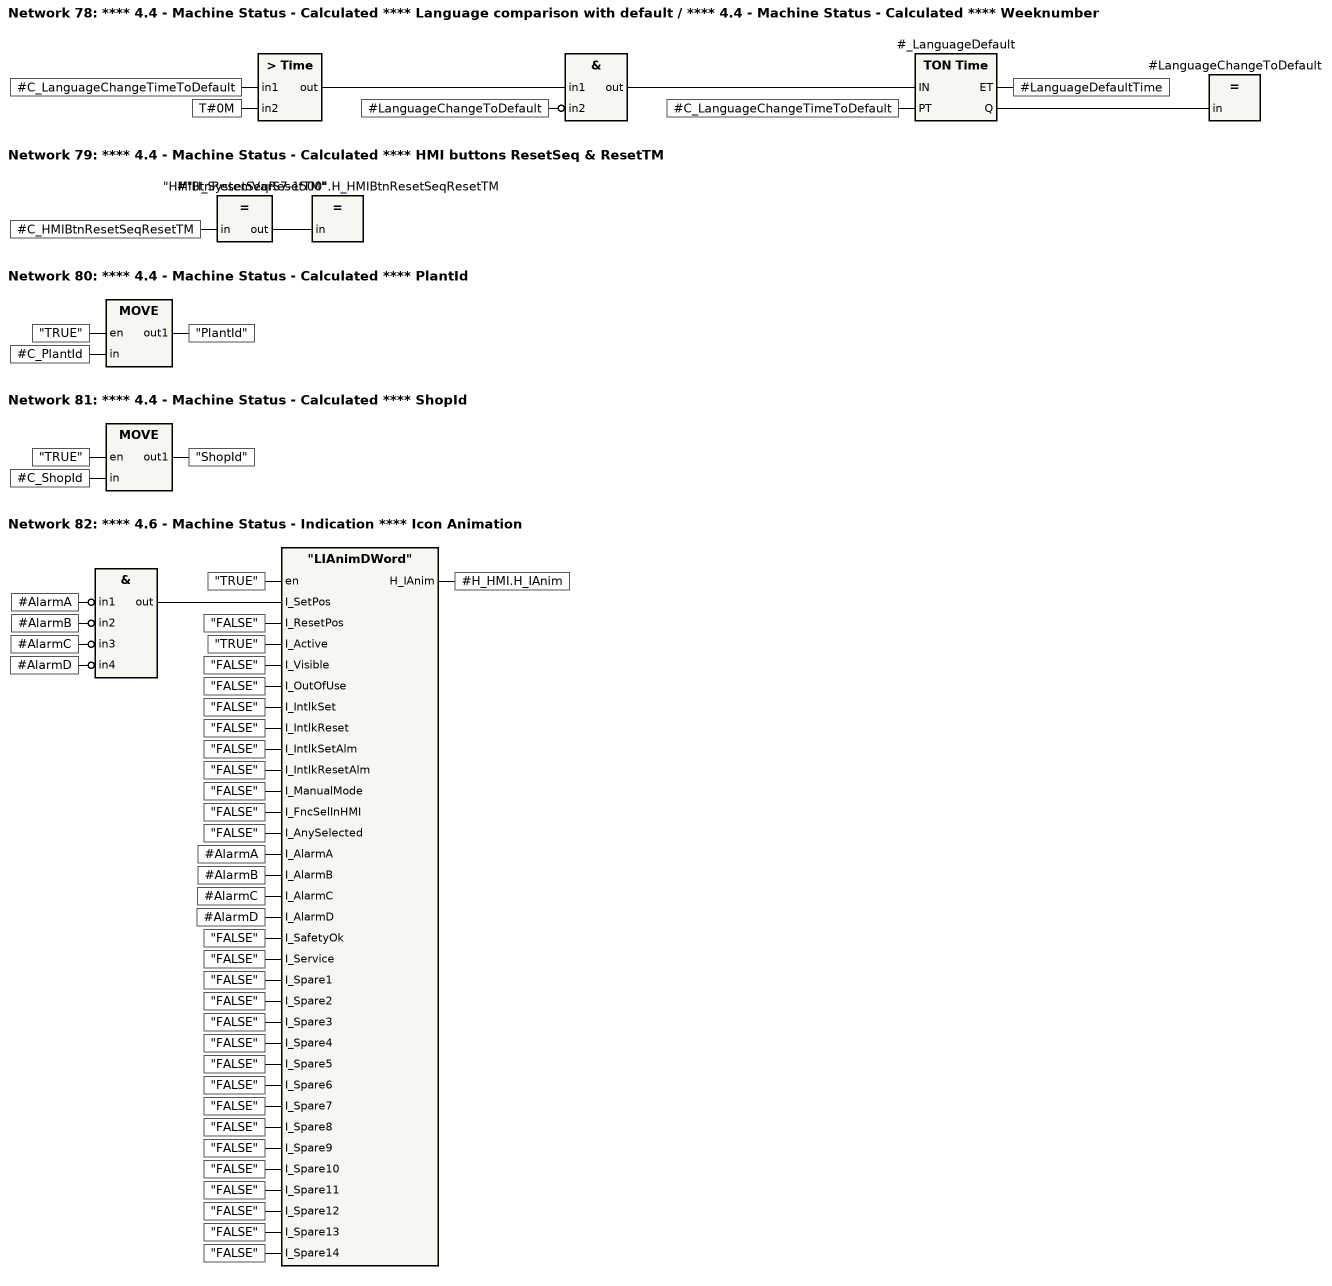
   #_LanguageDefault(IN := (#C_LanguageChangeTimeToDefault > T#0M) AND NOT #LanguageChangeToDefault,   // TON
                     PT := #C_LanguageChangeTimeToDefault,
                     ET => #LanguageDefaultTime);
   #LanguageChangeToDefault := #_LanguageDefault.Q;
END_REGION

REGION Network 79: **** 4.4 - Machine Status - Calculated **** HMI buttons ResetSeq & ResetTM
   // 0=Buttons are separate ; 1=Buttons are common
   "HMIBtnResetSeqResetTM" := #C_HMIBtnResetSeqResetTM;
   #"H_SystemVarS7-1500".H_HMIBtnResetSeqResetTM := #C_HMIBtnResetSeqResetTM;
END_REGION

REGION Network 80: **** 4.4 - Machine Status - Calculated **** PlantId
   IF "TRUE" THEN "PlantId" := #C_PlantId; END_IF;
END_REGION

REGION Network 81: **** 4.4 - Machine Status - Calculated **** ShopId
   IF "TRUE" THEN "ShopId" := #C_ShopId; END_IF;
END_REGION

REGION Network 82: **** 4.6 - Machine Status - Indication **** Icon Animation
   // Icon Animation
   IF "TRUE" THEN
       "LIAnimDWord"(I_SetPos := NOT #AlarmA AND NOT #AlarmB AND NOT #AlarmC AND NOT #AlarmD,
                     I_ResetPos := "FALSE",
                     I_Active := "TRUE",
                     I_Visible := "FALSE",
                     I_OutOfUse := "FALSE",
                     I_IntlkSet := "FALSE",
                     I_IntlkReset := "FALSE",
                     I_IntlkSetAlm := "FALSE",
                     I_IntlkResetAlm := "FALSE",
                     I_ManualMode := "FALSE",
                     I_FncSelInHMI := "FALSE",
                     I_AnySelected := "FALSE",
                     I_AlarmA := #AlarmA,
                     I_AlarmB := #AlarmB,
                     I_AlarmC := #AlarmC,
                     I_AlarmD := #AlarmD,
                     I_SafetyOk := "FALSE",
                     I_Service := "FALSE",
                     I_Spare1 := "FALSE",
                     I_Spare2 := "FALSE",
                     I_Spare3 := "FALSE",
                     I_Spare4 := "FALSE",
                     I_Spare5 := "FALSE",
                     I_Spare6 := "FALSE",
                     I_Spare7 := "FALSE",
                     I_Spare8 := "FALSE",
                     I_Spare9 := "FALSE",
                     I_Spare10 := "FALSE",
                     I_Spare11 := "FALSE",
                     I_Spare12 := "FALSE",
                     I_Spare13 := "FALSE",
                     I_Spare14 := "FALSE",
                     H_IAnim => #H_HMI.H_IAnim);
   END_IF;
END_REGION

REGION Network 83: **** 4.6 - Machine Status - Indication **** Animation
   // Animation
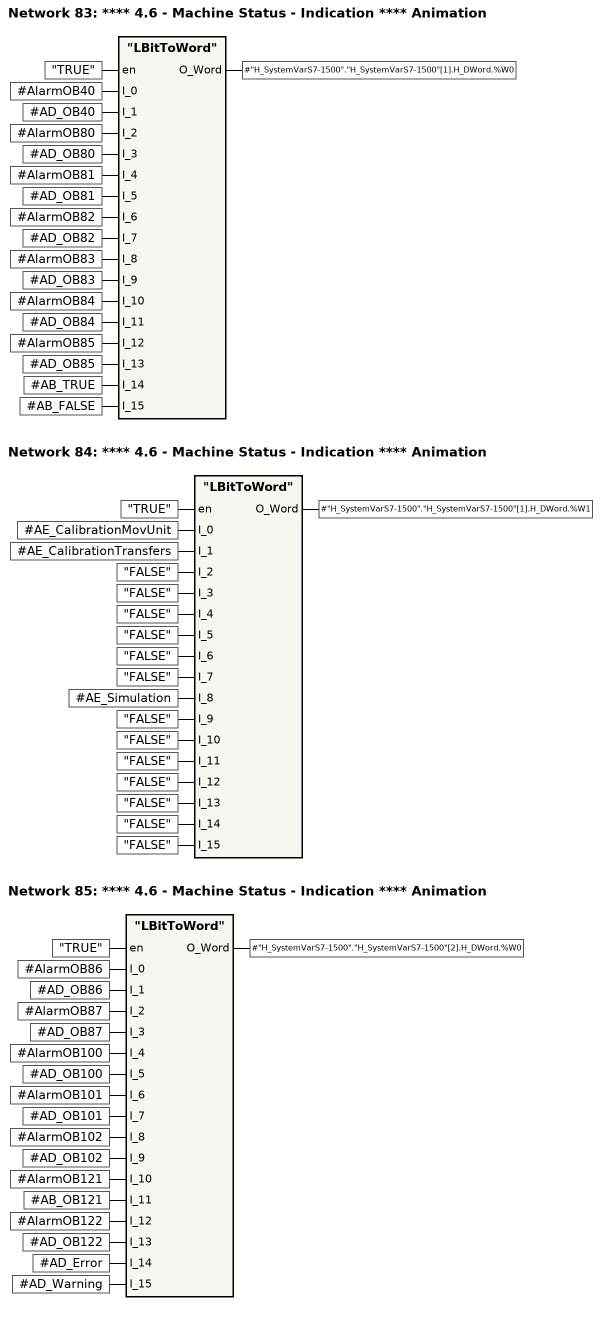
   IF "TRUE" THEN
       "LBitToWord"(I_0 := #AlarmOB40,
                    I_1 := #AD_OB40,
                    I_2 := #AlarmOB80,
                    I_3 := #AD_OB80,
                    I_4 := #AlarmOB81,
                    I_5 := #AD_OB81,
                    I_6 := #AlarmOB82,
                    I_7 := #AD_OB82,
                    I_8 := #AlarmOB83,
                    I_9 := #AD_OB83,
                    I_10 := #AlarmOB84,
                    I_11 := #AD_OB84,
                    I_12 := #AlarmOB85,
                    I_13 := #AD_OB85,
                    I_14 := #AB_TRUE,
                    I_15 := #AB_FALSE,
                    O_Word => #"H_SystemVarS7-1500"."H_SystemVarS7-1500"[1].H_DWord.%W0);
   END_IF;
END_REGION

REGION Network 84: **** 4.6 - Machine Status - Indication **** Animation
   // Animation
   IF "TRUE" THEN
       "LBitToWord"(I_0 := #AE_CalibrationMovUnit,
                    I_1 := #AE_CalibrationTransfers,
                    I_2 := "FALSE",
                    I_3 := "FALSE",
                    I_4 := "FALSE",
                    I_5 := "FALSE",
                    I_6 := "FALSE",
                    I_7 := "FALSE",
                    I_8 := #AE_Simulation,
                    I_9 := "FALSE",
                    I_10 := "FALSE",
                    I_11 := "FALSE",
                    I_12 := "FALSE",
                    I_13 := "FALSE",
                    I_14 := "FALSE",
                    I_15 := "FALSE",
                    O_Word => #"H_SystemVarS7-1500"."H_SystemVarS7-1500"[1].H_DWord.%W1);
   END_IF;
END_REGION

REGION Network 85: **** 4.6 - Machine Status - Indication **** Animation
   // Animation
   IF "TRUE" THEN
       "LBitToWord"(I_0 := #AlarmOB86,
                    I_1 := #AD_OB86,
                    I_2 := #AlarmOB87,
                    I_3 := #AD_OB87,
                    I_4 := #AlarmOB100,
                    I_5 := #AD_OB100,
                    I_6 := #AlarmOB101,
                    I_7 := #AD_OB101,
                    I_8 := #AlarmOB102,
                    I_9 := #AD_OB102,
                    I_10 := #AlarmOB121,
                    I_11 := #AB_OB121,
                    I_12 := #AlarmOB122,
                    I_13 := #AD_OB122,
                    I_14 := #AD_Error,
                    I_15 := #AD_Warning,
                    O_Word => #"H_SystemVarS7-1500"."H_SystemVarS7-1500"[2].H_DWord.%W0);
   END_IF;
END_REGION

REGION Network 86: **** 4.6 - Machine Status - Indication **** Animation
   // Animation
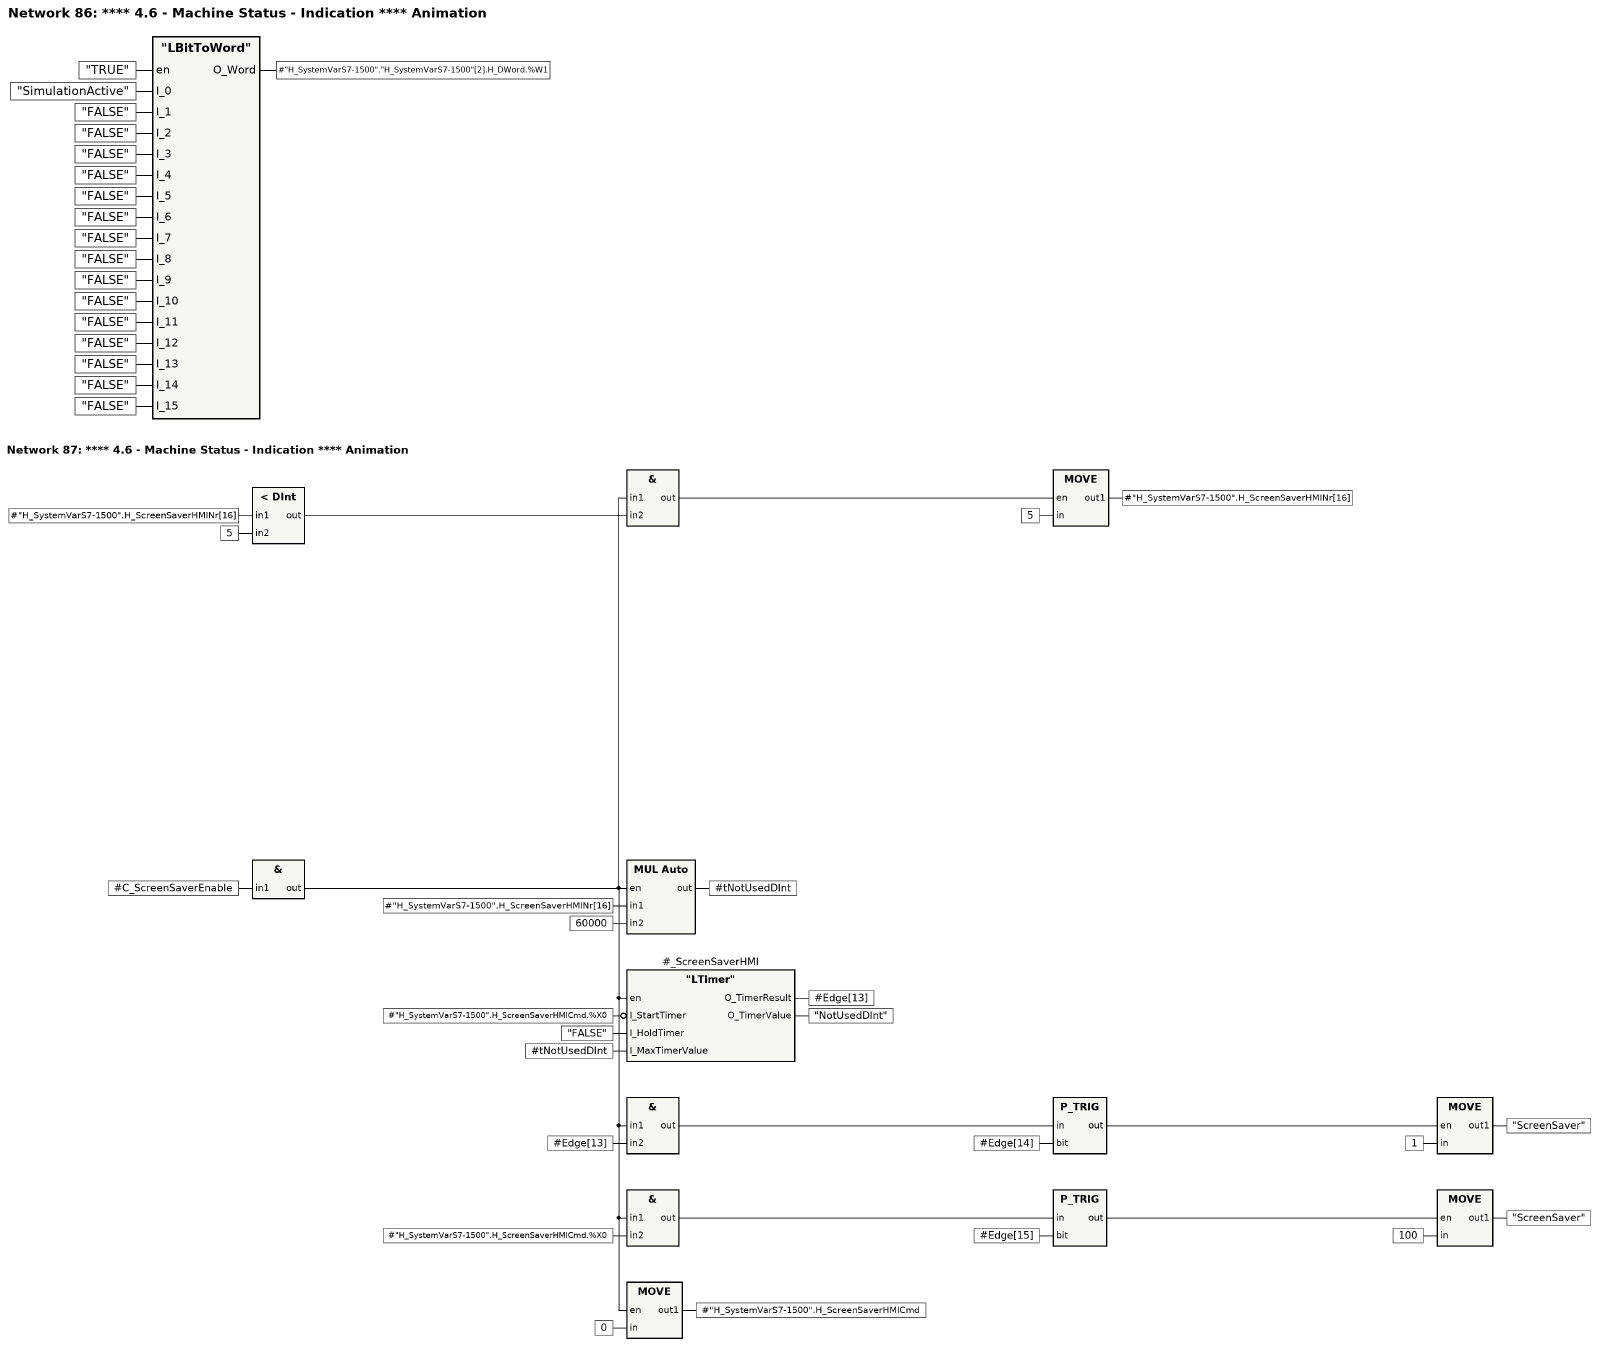
   IF "TRUE" THEN
       "LBitToWord"(I_0 := "SimulationActive",
                    I_1 := "FALSE",
                    I_2 := "FALSE",
                    I_3 := "FALSE",
                    I_4 := "FALSE",
                    I_5 := "FALSE",
                    I_6 := "FALSE",
                    I_7 := "FALSE",
                    I_8 := "FALSE",
                    I_9 := "FALSE",
                    I_10 := "FALSE",
                    I_11 := "FALSE",
                    I_12 := "FALSE",
                    I_13 := "FALSE",
                    I_14 := "FALSE",
                    I_15 := "FALSE",
                    O_Word => #"H_SystemVarS7-1500"."H_SystemVarS7-1500"[2].H_DWord.%W1);
   END_IF;
END_REGION

REGION Network 87: **** 4.6 - Machine Status - Indication **** Animation
   // Animation
   IF #C_ScreenSaverEnable AND (#"H_SystemVarS7-1500".H_ScreenSaverHMINr[16] < 5) THEN
       #"H_SystemVarS7-1500".H_ScreenSaverHMINr[16] := 5;
   END_IF;
   IF #C_ScreenSaverEnable THEN
       #tNotUsedDInt := #"H_SystemVarS7-1500".H_ScreenSaverHMINr[16] * 60000;
       #_ScreenSaverHMI(I_StartTimer := NOT #"H_SystemVarS7-1500".H_ScreenSaverHMICmd.%X0,   // "LTimer"
                        I_HoldTimer := "FALSE",
                        I_MaxTimerValue := #tNotUsedDInt,
                        O_TimerResult => #Edge[13],
                        O_TimerValue => "NotUsedDInt");
   END_IF;
   #_w1 := #C_ScreenSaverEnable AND #Edge[13];
   #_w2 := #_w1 AND NOT #Edge[14];   // rising edge
   #Edge[14] := #_w1;
   IF #_w2 THEN "ScreenSaver" := 1; END_IF;
   #_w3 := #C_ScreenSaverEnable AND #"H_SystemVarS7-1500".H_ScreenSaverHMICmd.%X0;
   #_w4 := #_w3 AND NOT #Edge[15];   // rising edge
   #Edge[15] := #_w3;
   IF #_w4 THEN "ScreenSaver" := 100; END_IF;
   IF #C_ScreenSaverEnable THEN #"H_SystemVarS7-1500".H_ScreenSaverHMICmd := 0; END_IF;
END_REGION

REGION Network 88: **** 4.6 - Machine Status - Indication **** Animation (LED status of the cpu)
   // Animation (LED status of the cpu)
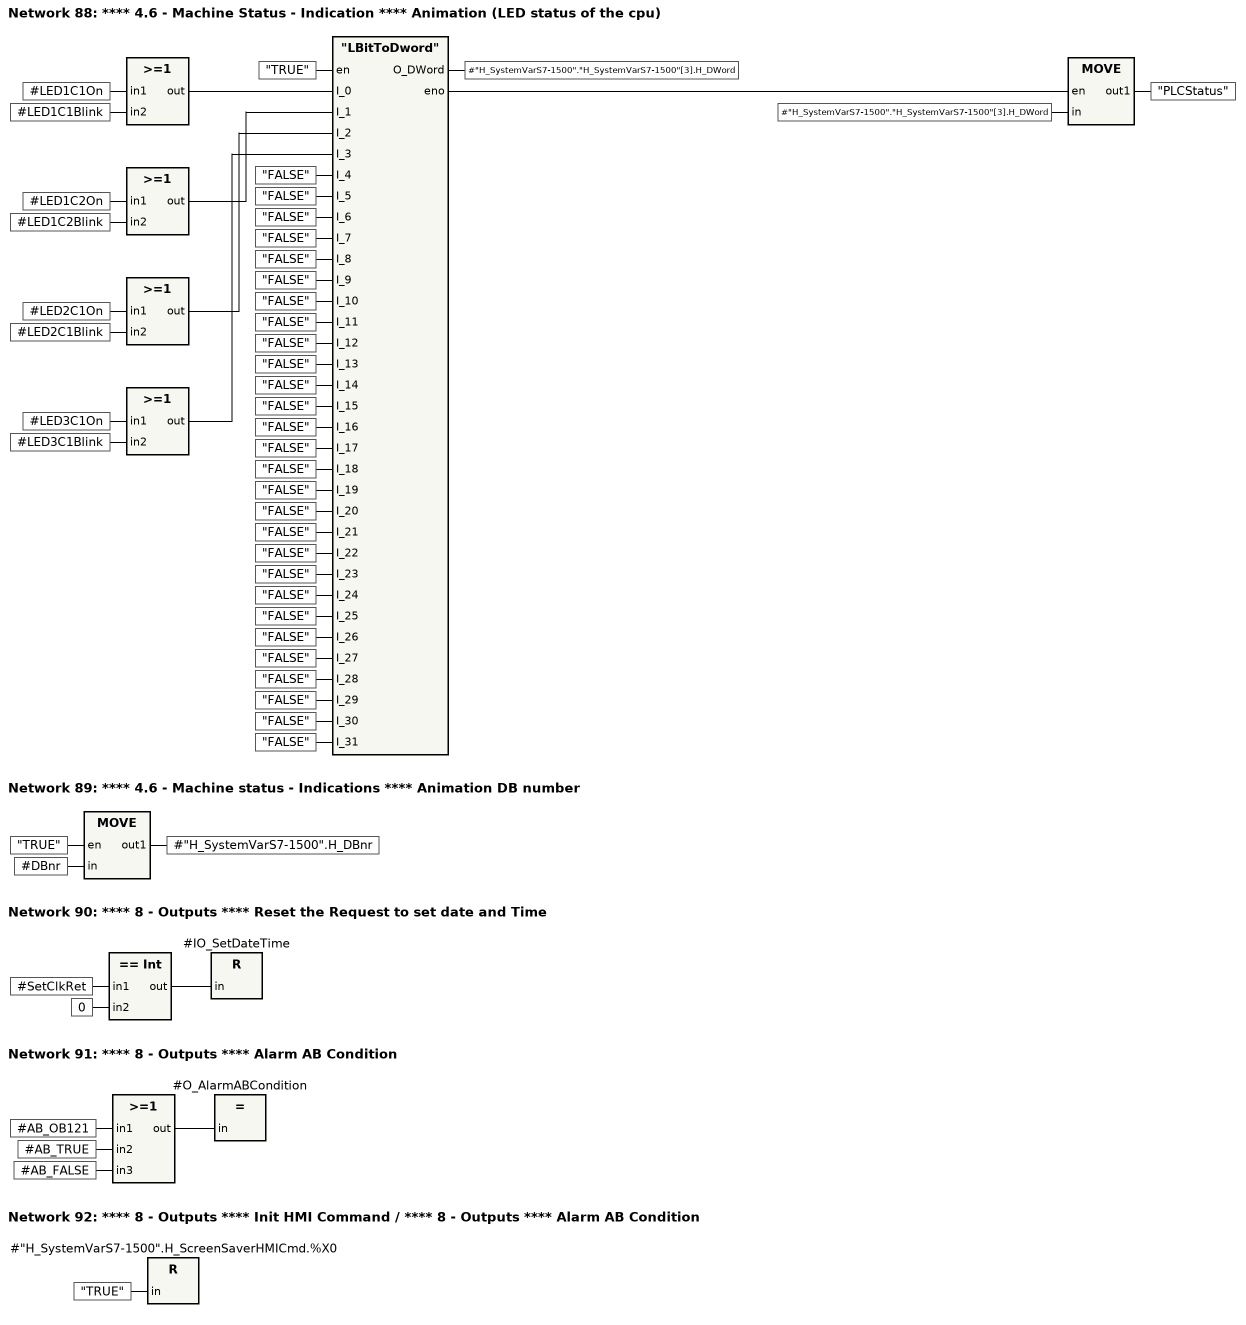
   "LBitToDword"(EN := "TRUE",
                 I_0 := #LED1C1On OR #LED1C1Blink,
                 I_1 := #LED1C2On OR #LED1C2Blink,
                 I_2 := #LED2C1On OR #LED2C1Blink,
                 I_3 := #LED3C1On OR #LED3C1Blink,
                 I_4 := "FALSE",
                 I_5 := "FALSE",
                 I_6 := "FALSE",
                 I_7 := "FALSE",
                 I_8 := "FALSE",
                 I_9 := "FALSE",
                 I_10 := "FALSE",
                 I_11 := "FALSE",
                 I_12 := "FALSE",
                 I_13 := "FALSE",
                 I_14 := "FALSE",
                 I_15 := "FALSE",
                 I_16 := "FALSE",
                 I_17 := "FALSE",
                 I_18 := "FALSE",
                 I_19 := "FALSE",
                 I_20 := "FALSE",
                 I_21 := "FALSE",
                 I_22 := "FALSE",
                 I_23 := "FALSE",
                 I_24 := "FALSE",
                 I_25 := "FALSE",
                 I_26 := "FALSE",
                 I_27 := "FALSE",
                 I_28 := "FALSE",
                 I_29 := "FALSE",
                 I_30 := "FALSE",
                 I_31 := "FALSE",
                 O_DWord => #"H_SystemVarS7-1500"."H_SystemVarS7-1500"[3].H_DWord,
                 ENO => #_w1);
   IF #_w1 THEN "PLCStatus" := #"H_SystemVarS7-1500"."H_SystemVarS7-1500"[3].H_DWord; END_IF;
END_REGION

REGION Network 89: **** 4.6 - Machine status - Indications **** Animation DB number
   // Animation DB number
   IF "TRUE" THEN #"H_SystemVarS7-1500".H_DBnr := #DBnr; END_IF;
END_REGION

REGION Network 90: **** 8 - Outputs **** Reset the Request to set date and Time
   // Reset the Request to set date and Time
   IF #SetClkRet = 0 THEN #IO_SetDateTime := FALSE; END_IF;
END_REGION

REGION Network 91: **** 8 - Outputs **** Alarm AB Condition
   // Alarm AB Condition
   #O_AlarmABCondition := #AB_OB121 OR #AB_TRUE OR #AB_FALSE;
END_REGION

REGION Network 92: **** 8 - Outputs **** Init HMI Command / **** 8 - Outputs **** Alarm AB Condition
   // Init HMI Command / Alarm AB Condition
   IF "TRUE" THEN #"H_SystemVarS7-1500".H_ScreenSaverHMICmd.%X0 := FALSE; END_IF;
END_REGION

REGION Network 93: **** 9 - Alarm Summary **** Alarm A
   // Alarm A
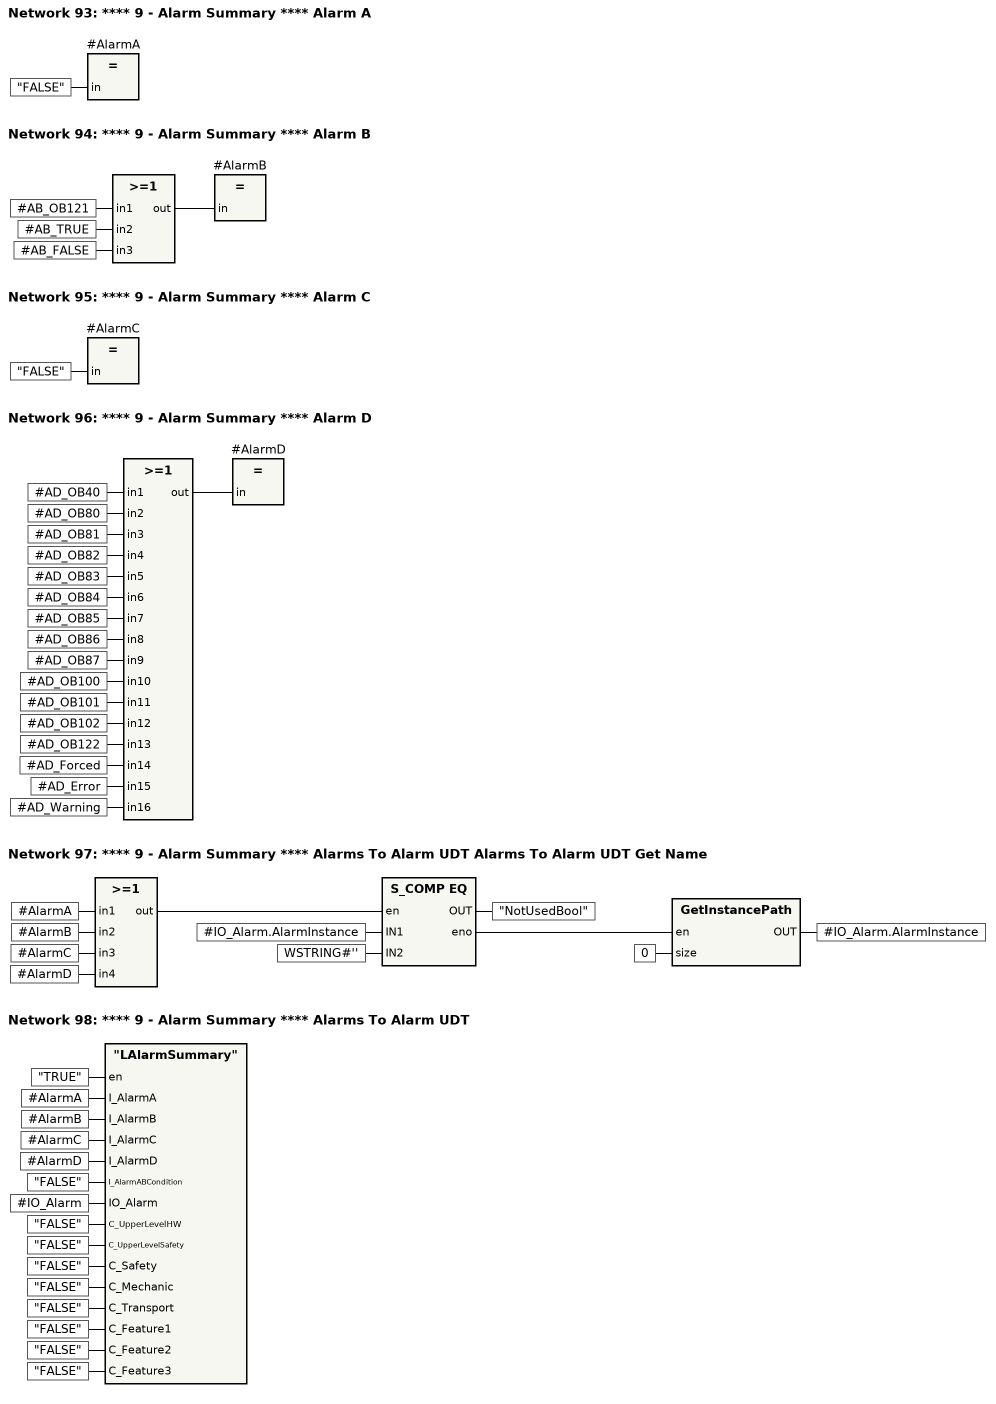
   #AlarmA := "FALSE";
END_REGION

REGION Network 94: **** 9 - Alarm Summary **** Alarm B
   // Alarm B
   #AlarmB := #AB_OB121 OR #AB_TRUE OR #AB_FALSE;
END_REGION

REGION Network 95: **** 9 - Alarm Summary **** Alarm C
   // Alarm C
   #AlarmC := "FALSE";
END_REGION

REGION Network 96: **** 9 - Alarm Summary **** Alarm D
   // Alarm D
   #AlarmD := #AD_OB40 OR #AD_OB80 OR #AD_OB81 OR #AD_OB82 OR #AD_OB83 OR #AD_OB84 OR #AD_OB85 OR #AD_OB86 OR #AD_OB87 OR #AD_OB100 OR #AD_OB101 OR #AD_OB102 OR #AD_OB122 OR #AD_Forced OR #AD_Error OR #AD_Warning;
END_REGION

REGION Network 97: **** 9 - Alarm Summary **** Alarms To Alarm UDT Alarms To Alarm UDT Get Name
   // Alarm / Alarm D
   S_COMP(EN := #AlarmA OR #AlarmB OR #AlarmC OR #AlarmD,
          IN1 := #IO_Alarm.AlarmInstance,
          IN2 := WSTRING#'',
          OUT => "NotUsedBool",
          ENO => #_w1);
   IF #_w1 THEN GetInstancePath(size := 0, OUT => #IO_Alarm.AlarmInstance); END_IF;
END_REGION

REGION Network 98: **** 9 - Alarm Summary **** Alarms To Alarm UDT
   // Alarm / Alarm D
   IF "TRUE" THEN
       "LAlarmSummary"(I_AlarmA := #AlarmA,
                       I_AlarmB := #AlarmB,
                       I_AlarmC := #AlarmC,
                       I_AlarmD := #AlarmD,
                       I_AlarmABCondition := "FALSE",
                       IO_Alarm := #IO_Alarm,
                       C_UpperLevelHW := "FALSE",
                       C_UpperLevelSafety := "FALSE",
                       C_Safety := "FALSE",
                       C_Mechanic := "FALSE",
                       C_Transport := "FALSE",
                       C_Feature1 := "FALSE",
                       C_Feature2 := "FALSE",
                       C_Feature3 := "FALSE");
   END_IF;
END_REGION

REGION Network 99: **** 9.1 - Alarm Output **** Alarm A
   // Alarm A
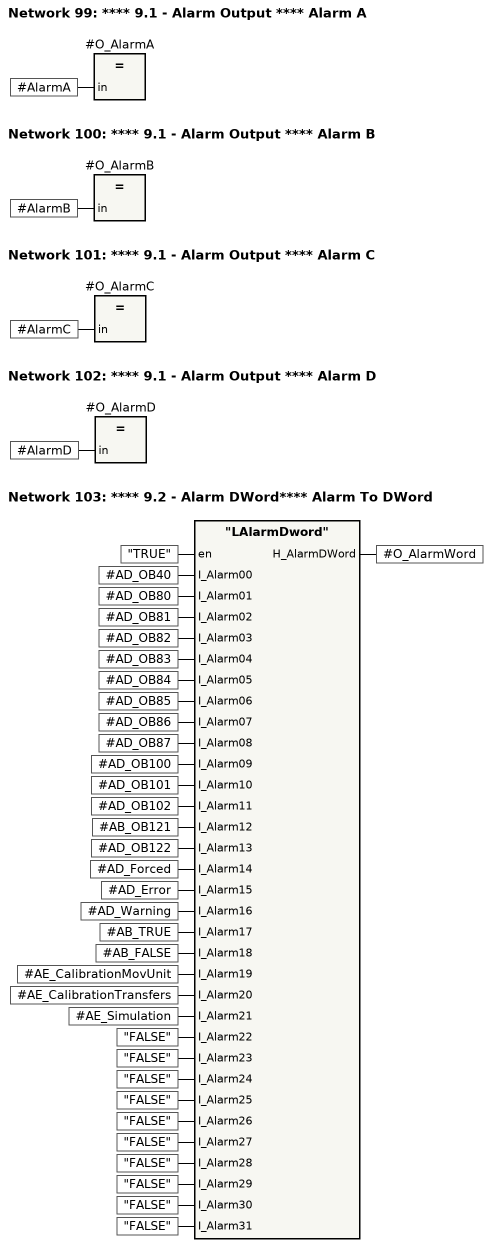
   #O_AlarmA := #AlarmA;
END_REGION

REGION Network 100: **** 9.1 - Alarm Output **** Alarm B
   // Alarm B
   #O_AlarmB := #AlarmB;
END_REGION

REGION Network 101: **** 9.1 - Alarm Output **** Alarm C
   // Alarm C
   #O_AlarmC := #AlarmC;
END_REGION

REGION Network 102: **** 9.1 - Alarm Output **** Alarm D
   // Alarm D
   #O_AlarmD := #AlarmD;
END_REGION

REGION Network 103: **** 9.2 - Alarm DWord**** Alarm To DWord
   // Alarm To Word
   IF "TRUE" THEN
       "LAlarmDword"(I_Alarm00 := #AD_OB40,
                     I_Alarm01 := #AD_OB80,
                     I_Alarm02 := #AD_OB81,
                     I_Alarm03 := #AD_OB82,
                     I_Alarm04 := #AD_OB83,
                     I_Alarm05 := #AD_OB84,
                     I_Alarm06 := #AD_OB85,
                     I_Alarm07 := #AD_OB86,
                     I_Alarm08 := #AD_OB87,
                     I_Alarm09 := #AD_OB100,
                     I_Alarm10 := #AD_OB101,
                     I_Alarm11 := #AD_OB102,
                     I_Alarm12 := #AB_OB121,
                     I_Alarm13 := #AD_OB122,
                     I_Alarm14 := #AD_Forced,
                     I_Alarm15 := #AD_Error,
                     I_Alarm16 := #AD_Warning,
                     I_Alarm17 := #AB_TRUE,
                     I_Alarm18 := #AB_FALSE,
                     I_Alarm19 := #AE_CalibrationMovUnit,
                     I_Alarm20 := #AE_CalibrationTransfers,
                     I_Alarm21 := #AE_Simulation,
                     I_Alarm22 := "FALSE",
                     I_Alarm23 := "FALSE",
                     I_Alarm24 := "FALSE",
                     I_Alarm25 := "FALSE",
                     I_Alarm26 := "FALSE",
                     I_Alarm27 := "FALSE",
                     I_Alarm28 := "FALSE",
                     I_Alarm29 := "FALSE",
                     I_Alarm30 := "FALSE",
                     I_Alarm31 := "FALSE",
                     H_AlarmDWord => #O_AlarmWord);
   END_IF;
END_REGION
END_FUNCTION_BLOCK
